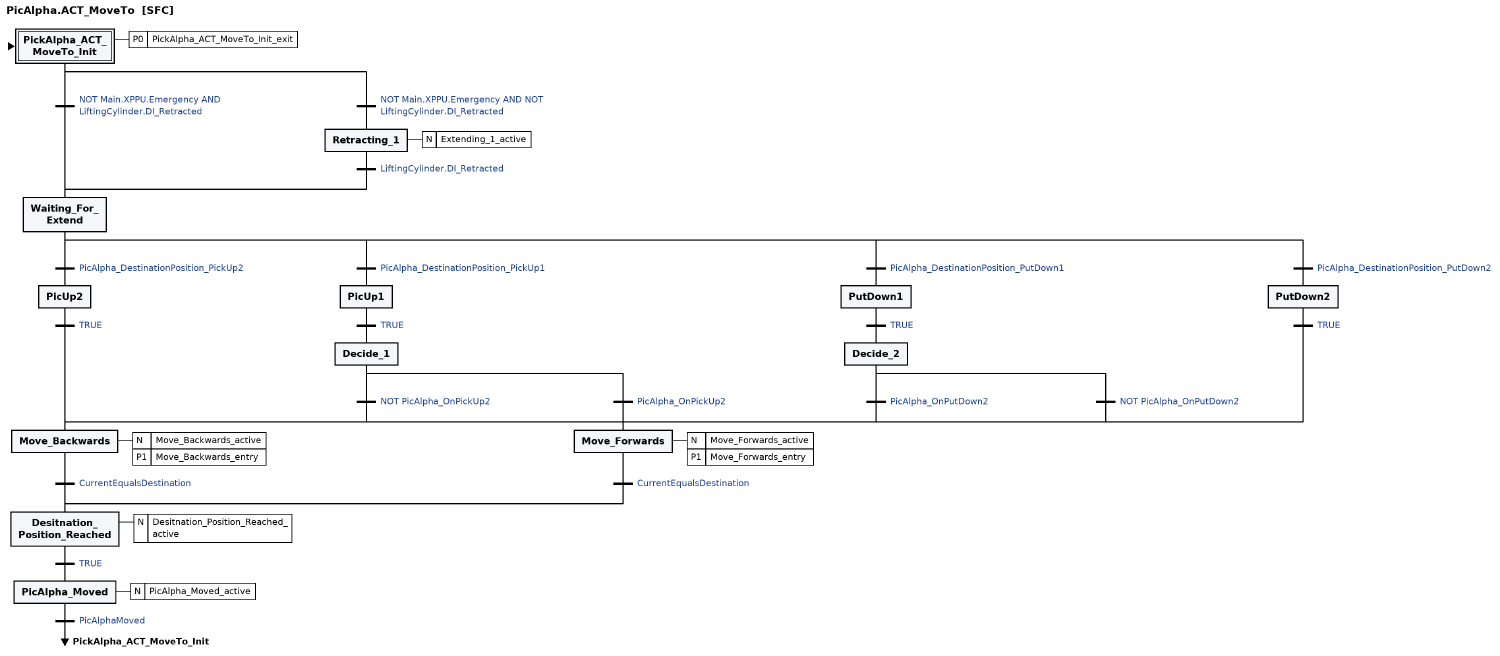
INITIAL_STEP PickAlpha_ACT_MoveTo_Init:
  PickAlpha_ACT_MoveTo_Init_exit(P0);
END_STEP
TRANSITION FROM PickAlpha_ACT_MoveTo_Init TO Waiting_For_Extend
  := NOT Main.XPPU.Emergency AND LiftingCylinder.DI_Retracted;
END_TRANSITION
TRANSITION FROM PickAlpha_ACT_MoveTo_Init TO Retracting_1
  := NOT Main.XPPU.Emergency AND NOT LiftingCylinder.DI_Retracted;
END_TRANSITION
STEP Retracting_1:
  Extending_1_active(N);
END_STEP
TRANSITION FROM Retracting_1 TO Waiting_For_Extend
  := LiftingCylinder.DI_Retracted;
END_TRANSITION
STEP Waiting_For_Extend:
END_STEP
TRANSITION FROM Waiting_For_Extend TO PicUp2
  := PicAlpha_DestinationPosition_PickUp2;
END_TRANSITION
TRANSITION FROM Waiting_For_Extend TO PicUp1
  := PicAlpha_DestinationPosition_PickUp1;
END_TRANSITION
TRANSITION FROM Waiting_For_Extend TO PutDown1
  := PicAlpha_DestinationPosition_PutDown1;
END_TRANSITION
TRANSITION FROM Waiting_For_Extend TO PutDown2
  := PicAlpha_DestinationPosition_PutDown2;
END_TRANSITION
STEP PicUp2:
END_STEP
TRANSITION FROM PicUp2 TO Move_Backwards
  := TRUE;
END_TRANSITION
STEP Move_Backwards:
  Move_Backwards_active(N);
  Move_Backwards_entry(P1);
END_STEP
TRANSITION FROM Move_Backwards TO Desitnation_Position_Reached
  := CurrentEqualsDestination;
END_TRANSITION
STEP PicUp1:
END_STEP
TRANSITION FROM PicUp1 TO Decide_1
  := TRUE;
END_TRANSITION
STEP Decide_1:
END_STEP
TRANSITION FROM Decide_1 TO Move_Backwards
  := NOT PicAlpha_OnPickUp2;
END_TRANSITION
TRANSITION FROM Decide_1 TO Move_Forwards
  := PicAlpha_OnPickUp2;
END_TRANSITION
STEP PutDown1:
END_STEP
TRANSITION FROM PutDown1 TO Decide_2
  := TRUE;
END_TRANSITION
STEP Decide_2:
END_STEP
TRANSITION FROM Decide_2 TO Move_Backwards
  := PicAlpha_OnPutDown2;
END_TRANSITION
TRANSITION FROM Decide_2 TO Move_Forwards
  := NOT PicAlpha_OnPutDown2;
END_TRANSITION
STEP PutDown2:
END_STEP
TRANSITION FROM PutDown2 TO Move_Forwards
  := TRUE;
END_TRANSITION
STEP Move_Forwards:
  Move_Forwards_active(N);
  Move_Forwards_entry(P1);
END_STEP
TRANSITION FROM Move_Forwards TO Desitnation_Position_Reached
  := CurrentEqualsDestination;
END_TRANSITION
STEP Desitnation_Position_Reached:
  Desitnation_Position_Reached_active(N);
END_STEP
TRANSITION FROM Desitnation_Position_Reached TO PicAlpha_Moved
  := TRUE;
END_TRANSITION
STEP PicAlpha_Moved:
  PicAlpha_Moved_active(N);
END_STEP
TRANSITION FROM PicAlpha_Moved TO PickAlpha_ACT_MoveTo_Init
  := PicAlphaMoved;
END_TRANSITION
END_ACTION

ACTION ACT_EmergencyStop:
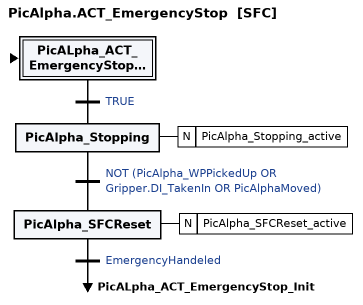
INITIAL_STEP PicALpha_ACT_EmergencyStop_Init:
END_STEP
TRANSITION FROM PicALpha_ACT_EmergencyStop_Init TO PicAlpha_Stopping
  := TRUE;
END_TRANSITION
STEP PicAlpha_Stopping:
  PicAlpha_Stopping_active(N);
END_STEP
TRANSITION FROM PicAlpha_Stopping TO PicAlpha_SFCReset
  := NOT (PicAlpha_WPPickedUp OR Gripper.DI_TakenIn OR PicAlphaMoved);
END_TRANSITION
STEP PicAlpha_SFCReset:
  PicAlpha_SFCReset_active(N);
END_STEP
TRANSITION FROM PicAlpha_SFCReset TO PicALpha_ACT_EmergencyStop_Init
  := EmergencyHandeled;
END_TRANSITION
END_ACTION

ACTION ACT_Init:
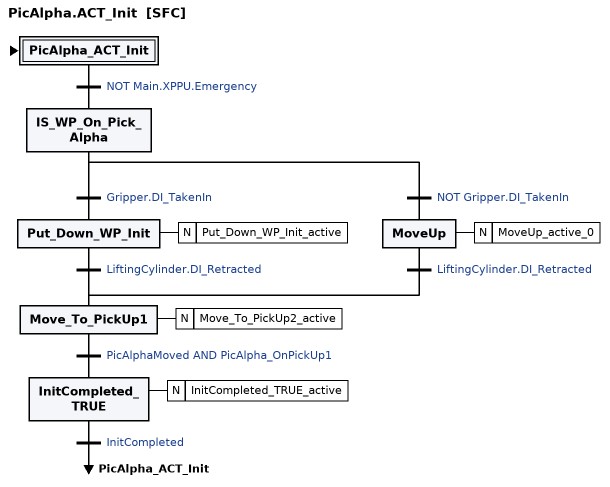
INITIAL_STEP PicAlpha_ACT_Init:
END_STEP
TRANSITION FROM PicAlpha_ACT_Init TO IS_WP_On_Pick_Alpha
  := NOT Main.XPPU.Emergency;
END_TRANSITION
STEP IS_WP_On_Pick_Alpha:
END_STEP
TRANSITION FROM IS_WP_On_Pick_Alpha TO Put_Down_WP_Init
  := Gripper.DI_TakenIn;
END_TRANSITION
TRANSITION FROM IS_WP_On_Pick_Alpha TO MoveUp
  := NOT Gripper.DI_TakenIn;
END_TRANSITION
STEP Put_Down_WP_Init:
  Put_Down_WP_Init_active(N);
END_STEP
TRANSITION FROM Put_Down_WP_Init TO Move_To_PickUp1
  := LiftingCylinder.DI_Retracted;
END_TRANSITION
STEP MoveUp:
  MoveUp_active_0(N);
END_STEP
TRANSITION FROM MoveUp TO Move_To_PickUp1
  := LiftingCylinder.DI_Retracted;
END_TRANSITION
STEP Move_To_PickUp1:
  Move_To_PickUp2_active(N);
END_STEP
TRANSITION FROM Move_To_PickUp1 TO InitCompleted_TRUE
  := PicAlphaMoved AND PicAlpha_OnPickUp1;
END_TRANSITION
STEP InitCompleted_TRUE:
  InitCompleted_TRUE_active(N);
END_STEP
TRANSITION FROM InitCompleted_TRUE TO PicAlpha_ACT_Init
  := InitCompleted;
END_TRANSITION
END_ACTION

ACTION ACT_AutomaticExecute:
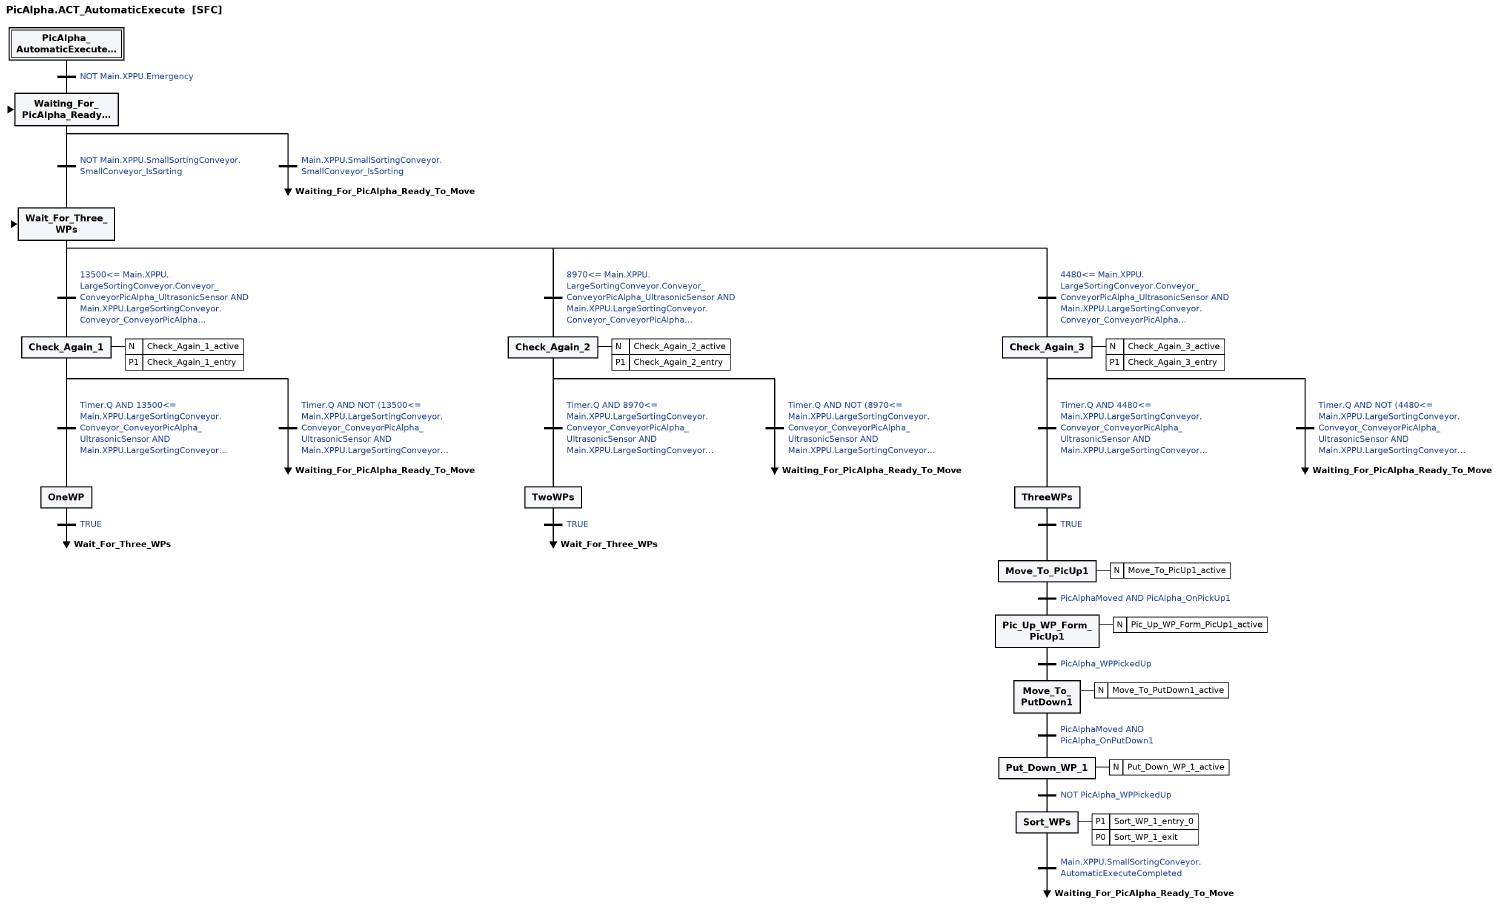
INITIAL_STEP PicAlpha_AutomaticExecute_Init:
END_STEP
TRANSITION FROM PicAlpha_AutomaticExecute_Init TO Waiting_For_PicAlpha_Ready_To_Move
  := NOT Main.XPPU.Emergency;
END_TRANSITION
STEP Waiting_For_PicAlpha_Ready_To_Move:
END_STEP
TRANSITION FROM Waiting_For_PicAlpha_Ready_To_Move TO Wait_For_Three_WPs
  := NOT Main.XPPU.SmallSortingConveyor.SmallConveyor_IsSorting;
END_TRANSITION
TRANSITION FROM Waiting_For_PicAlpha_Ready_To_Move TO Waiting_For_PicAlpha_Ready_To_Move
  := Main.XPPU.SmallSortingConveyor.SmallConveyor_IsSorting;
END_TRANSITION
STEP Wait_For_Three_WPs:
END_STEP
TRANSITION FROM Wait_For_Three_WPs TO Check_Again_1
  := 13500<= Main.XPPU.LargeSortingConveyor.Conveyor_ConveyorPicAlpha_UltrasonicSensor AND Main.XPPU.LargeSortingConveyor.Conveyor_ConveyorPicAlpha_UltrasonicSensor<=13700;
END_TRANSITION
TRANSITION FROM Wait_For_Three_WPs TO Check_Again_2
  := 8970<= Main.XPPU.LargeSortingConveyor.Conveyor_ConveyorPicAlpha_UltrasonicSensor AND Main.XPPU.LargeSortingConveyor.Conveyor_ConveyorPicAlpha_UltrasonicSensor<=9170;
END_TRANSITION
TRANSITION FROM Wait_For_Three_WPs TO Check_Again_3
  := 4480<= Main.XPPU.LargeSortingConveyor.Conveyor_ConveyorPicAlpha_UltrasonicSensor AND Main.XPPU.LargeSortingConveyor.Conveyor_ConveyorPicAlpha_UltrasonicSensor<=4680;
END_TRANSITION
STEP Check_Again_1:
  Check_Again_1_active(N);
  Check_Again_1_entry(P1);
END_STEP
TRANSITION FROM Check_Again_1 TO OneWP
  := Timer.Q AND 13500<= Main.XPPU.LargeSortingConveyor.Conveyor_ConveyorPicAlpha_UltrasonicSensor AND Main.XPPU.LargeSortingConveyor.Conveyor_ConveyorPicAlpha_UltrasonicSensor<=13700;
END_TRANSITION
TRANSITION FROM Check_Again_1 TO Waiting_For_PicAlpha_Ready_To_Move
  := Timer.Q AND NOT (13500<= Main.XPPU.LargeSortingConveyor.Conveyor_ConveyorPicAlpha_UltrasonicSensor AND Main.XPPU.LargeSortingConveyor.Conveyor_ConveyorPicAlpha_UltrasonicSensor<=13700);
END_TRANSITION
STEP OneWP:
END_STEP
TRANSITION FROM OneWP TO Wait_For_Three_WPs
  := TRUE;
END_TRANSITION
STEP Check_Again_2:
  Check_Again_2_active(N);
  Check_Again_2_entry(P1);
END_STEP
TRANSITION FROM Check_Again_2 TO TwoWPs
  := Timer.Q AND 8970<= Main.XPPU.LargeSortingConveyor.Conveyor_ConveyorPicAlpha_UltrasonicSensor AND Main.XPPU.LargeSortingConveyor.Conveyor_ConveyorPicAlpha_UltrasonicSensor<=9170;
END_TRANSITION
TRANSITION FROM Check_Again_2 TO Waiting_For_PicAlpha_Ready_To_Move
  := Timer.Q AND NOT (8970<= Main.XPPU.LargeSortingConveyor.Conveyor_ConveyorPicAlpha_UltrasonicSensor AND Main.XPPU.LargeSortingConveyor.Conveyor_ConveyorPicAlpha_UltrasonicSensor<=9170);
END_TRANSITION
STEP TwoWPs:
END_STEP
TRANSITION FROM TwoWPs TO Wait_For_Three_WPs
  := TRUE;
END_TRANSITION
STEP Check_Again_3:
  Check_Again_3_active(N);
  Check_Again_3_entry(P1);
END_STEP
TRANSITION FROM Check_Again_3 TO ThreeWPs
  := Timer.Q AND 4480<= Main.XPPU.LargeSortingConveyor.Conveyor_ConveyorPicAlpha_UltrasonicSensor AND Main.XPPU.LargeSortingConveyor.Conveyor_ConveyorPicAlpha_UltrasonicSensor<=4680;
END_TRANSITION
TRANSITION FROM Check_Again_3 TO Waiting_For_PicAlpha_Ready_To_Move
  := Timer.Q AND NOT (4480<= Main.XPPU.LargeSortingConveyor.Conveyor_ConveyorPicAlpha_UltrasonicSensor AND Main.XPPU.LargeSortingConveyor.Conveyor_ConveyorPicAlpha_UltrasonicSensor<=4680);
END_TRANSITION
STEP ThreeWPs:
END_STEP
TRANSITION FROM ThreeWPs TO Move_To_PicUp1
  := TRUE;
END_TRANSITION
STEP Move_To_PicUp1:
  Move_To_PicUp1_active(N);
END_STEP
TRANSITION FROM Move_To_PicUp1 TO Pic_Up_WP_Form_PicUp1
  := PicAlphaMoved AND PicAlpha_OnPickUp1;
END_TRANSITION
STEP Pic_Up_WP_Form_PicUp1:
  Pic_Up_WP_Form_PicUp1_active(N);
END_STEP
TRANSITION FROM Pic_Up_WP_Form_PicUp1 TO Move_To_PutDown1
  := PicAlpha_WPPickedUp;
END_TRANSITION
STEP Move_To_PutDown1:
  Move_To_PutDown1_active(N);
END_STEP
TRANSITION FROM Move_To_PutDown1 TO Put_Down_WP_1
  := PicAlphaMoved AND PicAlpha_OnPutDown1;
END_TRANSITION
STEP Put_Down_WP_1:
  Put_Down_WP_1_active(N);
END_STEP
TRANSITION FROM Put_Down_WP_1 TO Sort_WPs
  := NOT PicAlpha_WPPickedUp;
END_TRANSITION
STEP Sort_WPs:
  Sort_WP_1_entry_0(P1);
  Sort_WP_1_exit(P0);
END_STEP
TRANSITION FROM Sort_WPs TO Waiting_For_PicAlpha_Ready_To_Move
  := Main.XPPU.SmallSortingConveyor.AutomaticExecuteCompleted;
END_TRANSITION
END_ACTION

ACTION Sort_WP_1_active:
                      Main.XPPU.SmallSortingConveyor.ACT_SortWP();
                    
END_ACTION

ACTION Sort_WP_3_entry_0:
                      SC_PicAlpha_AllowToOperate:=TRUE;
                    
END_ACTION

ACTION Extending_active:
                      LiftingCylinder.ACT_Extend();
                    
END_ACTION

ACTION Check_Again_1_entry:
                      Timer(IN:=FALSE);
                    
END_ACTION

ACTION Move_Forwards_active:
                      Motor.ACT_TurnForwards();
IF(PicAlpha_DestinationPosition_PickUp2=PicAlpha_OnPickUp2 AND PicAlpha_OnPickUp2)THEN
	CurrentEqualsDestination:=TRUE;
ELSIF(PicAlpha_DestinationPosition_PutDown1=PicAlpha_OnPutDown1 AND PicAlpha_OnPutDown1 )THEN
	CurrentEqualsDestination:=TRUE;	
ELSIF(PicAlpha_DestinationPosition_PutDown2=PicAlpha_OnPutDown2 AND PicAlpha_OnPutDown2)THEN
	CurrentEqualsDestination:=TRUE;
END_IF
                    
END_ACTION

ACTION Desitnation_Position_Reached_active:
                      Motor.ACT_Stop();
                    
END_ACTION

ACTION Sort_WP_2_entry:
                      Main.XPPU.SmallSortingConveyor.HelpACT_WPSorted_FALSE();
                    
END_ACTION

ACTION Sort_WP_3_entry:
                      Main.XPPU.SmallSortingConveyor.HelpACT_WPSorted_FALSE();
                    
END_ACTION

ACTION PickAlpha_ACT_MoveTo_Init_exit:
                      PicAlphaMoved:=FALSE;
                    
END_ACTION

ACTION Sort_WP_2_active:
                      Main.XPPU.SmallSortingConveyor.ACT_SortWP();
                    
END_ACTION

ACTION Seperate_First_WP_active:
                      Main.XPPU.ConveyorPicAlpha.ACT_SeperateWP();
                    
END_ACTION

ACTION Move_To_PicUp1_active:
                      PicAlpha_DestinationPosition_PickUp1:=TRUE;
PicAlpha_DestinationPosition_PickUp2:=FALSE;
PicAlpha_DestinationPosition_PutDown1:=FALSE;
PicAlpha_DestinationPosition_PutDown2:=FALSE;
ACT_MoveTo();
                    
END_ACTION

ACTION MoveUp_active:
                      LiftingCylinder.ACT_Retract();
                    
END_ACTION

ACTION Move_Backwards_entry:
                      CurrentEqualsDestination:=FALSE;
                    
END_ACTION

ACTION Extending_1_active:
                      LiftingCylinder.ACT_Retract();
                    
END_ACTION

ACTION Retracting_PicAlpha_exit:
                      PicAlpha_WPPickedUp:=TRUE;
                    
END_ACTION

ACTION Sort_WP_2_exit:
                      SC_PicAlpha_AllowToOperate:=FALSE;
                    
END_ACTION

ACTION Sort_WP_3_exit:
                      SC_PicAlpha_AllowToOperate:=FALSE;
                    
END_ACTION

ACTION Sort_WP_2_entry_0:
                      SC_PicAlpha_AllowToOperate:=TRUE;
                    
END_ACTION

ACTION Pic_Up_WP_Form_PicUp1_active:
                      ACT_PickUpWP();
                    
END_ACTION

ACTION PicAlpha_Moved_active:
                      PicAlphaMoved:=TRUE;
                    
END_ACTION

ACTION Put_Down_WP_Init_active:
                      ACT_PutDownWP();
                    
END_ACTION

ACTION Extending_PicUp_active:
                      LiftingCylinder.ACT_Extend();
                    
END_ACTION

ACTION Check_Again_3_entry:
                      Timer(IN:=FALSE);
                    
END_ACTION

ACTION Error_active:
                      LiftingCylinder.ACT_Retract();
PicAlpha_SoftwareEmergency:=true;
                    
END_ACTION

ACTION Put_Down_WP_1_active:
                      ACT_PutDownWP();
                    
END_ACTION

ACTION Sort_WP_3_active:
                      Main.XPPU.SmallSortingConveyor.ACT_SortWP();
                    
END_ACTION

ACTION Check_Again_2_active:
                      Timer(IN:=TRUE, PT:=T#500ms);
                    
END_ACTION

ACTION Sort_WP_1_entry:
                      SC_PicAlpha_AllowToOperate:=TRUE;
                    
END_ACTION

ACTION Step0_ACT_EmergencyStop_active:
                      SFCReset:=TRUE;
                    
END_ACTION

ACTION Sort_WP_1_entry_0:
                      SC_PicAlpha_AllowToOperate:=TRUE;
                    
END_ACTION

ACTION Check_Again_3_active:
                      Timer(IN:=TRUE, PT:=T#500ms);
                    
END_ACTION

ACTION Retracting_active:
                      PicAlphaVacuumHit:=FALSE;
LiftingCylinder.ACT_Retract();
                    
END_ACTION

ACTION Move_Forwards_entry:
                      CurrentEqualsDestination:=FALSE;
                    
END_ACTION

ACTION Seperate_First_WP_entry:
                      //Main.XPPU.ConveyorPicALpha.HelpACT_WPSeperated_FALSE();
                    
END_ACTION

ACTION MoveUp_entry:
                      Timer(IN:=FALSE);
                    
END_ACTION

ACTION Retracting_exit:
                      PicAlpha_WPPickedUp:=FALSE;
                    
END_ACTION

ACTION Stop_Vacuum_active:
                      Gripper.ACT_Release();
PicAlphaVacuumHit:=TRUE;
                    
END_ACTION

ACTION Check_Again_1_active:
                      Timer(IN:=TRUE, PT:=T#500ms);
                    
END_ACTION

ACTION InitCompleted_FALSE_active:
                      InitCompleted:=FALSE;
                    
END_ACTION

ACTION Intaking_PicUp_active:
                      Gripper.ACT_Intake();
Timer(IN:=true, PT:=T#2s);
                    
END_ACTION

ACTION Retracting_PicAlpha_active:
                      LiftingCylinder.ACT_Retract();
                    
END_ACTION

ACTION PicAlpha_Stopping_active:
                      PicAlpha_WPPickedUp:=FALSE;
PicAlpha_DestinationPosition_PickUp1:=FALSE;
PicAlpha_DestinationPosition_PickUp2:=FALSE;
PicAlpha_DestinationPosition_PutDown1:=FALSE;
PicAlpha_DestinationPosition_PutDown2:=FALSE;

Gripper.ACT_Release();
PicAlphaVacuumHit:=FALSE;	
Motor.ACT_Stop();

CurrentEqualsDestination:=FALSE;
PicAlphaMoved:=FALSE;
                    
END_ACTION

ACTION PicAlpha_SFCReset_active:
                       EmergencyHandeled:=TRUE;	
                    
END_ACTION

ACTION Move_To_PutDown1_active:
                      PicAlpha_DestinationPosition_PickUp1:=FALSE;
PicAlpha_DestinationPosition_PickUp2:=FALSE;
PicAlpha_DestinationPosition_PutDown1:=TRUE;
PicAlpha_DestinationPosition_PutDown2:=FALSE;
ACT_MoveTo();
                    
END_ACTION

ACTION Seperate_Second_WP_entry:
                      //Main.XPPU.ConveyorPicALpha.HelpACT_WPSeperated_FALSE();
                    
END_ACTION

ACTION Intaking_PicUp_entry:
                      Timer(IN:=FALSE);
                    
END_ACTION

ACTION MoveUp_active_0:
                      LiftingCylinder.ACT_Retract();
                    
END_ACTION

ACTION Sort_WP_1_exit:
                      SC_PicAlpha_AllowToOperate:=FALSE;
                    
END_ACTION

ACTION InitCompleted_TRUE_active:
                      InitCompleted:=TRUE;
                    
END_ACTION

ACTION PicAlpha_StopVacuum_active:
                      Gripper.ACT_Release();
                    
END_ACTION

ACTION Seperate_Second_WP_active:
                      Main.XPPU.ConveyorPicAlpha.ACT_SeperateWP();
                    
END_ACTION

ACTION Move_Backwards_active:
                      Motor.ACT_TurnBackwards();
CurrentEqualsDestination:=FALSE;
IF(PicAlpha_DestinationPosition_PickUp1=PicAlpha_OnPickUp1 AND PicAlpha_OnPickUp1)THEN
	CurrentEqualsDestination:=TRUE;
ELSIF(PicAlpha_DestinationPosition_PickUp2=PicAlpha_OnPickUp2 AND PicAlpha_OnPickUp2)THEN
	CurrentEqualsDestination:=TRUE;
ELSIF(PicAlpha_DestinationPosition_PutDown1=PicAlpha_OnPutDown1 AND PicAlpha_OnPutDown1)THEN
	CurrentEqualsDestination:=TRUE;	
END_IF
                    
END_ACTION

ACTION Check_Again_2_entry:
                      Timer(IN:=FALSE);
                    
END_ACTION

ACTION Move_To_PickUp2_active:
                      PicAlpha_DestinationPosition_PickUp1:=TRUE;
PicAlpha_DestinationPosition_PickUp2:=FALSE;
PicAlpha_DestinationPosition_PutDown1:=FALSE;
PicAlpha_DestinationPosition_PutDown2:=FALSE;

ACT_MoveTo();
                    
END_ACTION
END_FUNCTION_BLOCK

FUNCTION_BLOCK SeperatorConveyor_Refill
VAR_INPUT	
	SwitchStopper : Switch;
	Motor : Motor;
	//Software	
	SFCReset : BOOL;
	InitCompleted : BOOL;
	LSC_AllowedToOperate : BOOL;
	AutomaticExecuteReceivingCompleted : BOOL;
	EmergencyHandeled : BOOL;
END_VAR
VAR_OUTPUT	
	//Software	
	SeperatorConveyor_WPSeperated : BOOL;
	SeperatorConveyor_IsRefilling : BOOL;
	SeperatorConveyor_RefillingIsActive : BOOL;
	SeperatorConveyor_NumberOfWPs : INT;
END_VAR
VAR
	//Hardware
	SeperaterConveyor_Beginning_PresenceSensor AT %I* : BOOL;
	SeperaterConveyor_End_PresenceSensor AT %I* : BOOL;
	
	//Software
	Timer:TON;
END_VAR

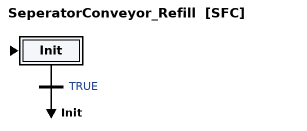
INITIAL_STEP Init:
END_STEP
TRANSITION FROM Init TO Init
  := TRUE;
END_TRANSITION

ACTION Turn_On_Conveyor_entry:
                      Timer(IN:=FALSE);
                    
END_ACTION

ACTION HelpACT_WPSeperated_FALSE:
                      SeperatorConveyor_WPSeperated:=FALSE;
                    
END_ACTION

ACTION TurnForwards_PAC_entry:
                      Timer(IN:=FALSE);
                    
END_ACTION

ACTION Turn_Off_Conveyor_active_0:
                      Motor.ACT_Stop();
                    
END_ACTION

ACTION Stop_PAC_active:
                      Motor.ACT_Stop();
                    
END_ACTION

ACTION Turn_On_Conveyor_active:
                      Motor.ACT_TurnForwards();

Timer(IN:=TRUE, PT:=T#500ms);
	
                    
END_ACTION

ACTION Refilling_LargeSortingConveyor_entry:
                      SeperatorConveyor_IsRefilling:=TRUE;
SeperatorConveyor_RefillingIsActive:=TRUE;
                    
END_ACTION

ACTION SeperaterConveyor_SFCReset_active:
                      EmergencyHandeled:=TRUE;		
                    
END_ACTION

ACTION Stop_Conveyor_active:
                      Motor.ACT_Stop();	
                    
END_ACTION

ACTION Trun_Forwards_AE_entry:
                      Timer(IN:=FALSE);
                    
END_ACTION

ACTION Sort_WP_active_0:
                      Main.XPPU.LargeSortingConveyor.ACT_SortWP();
                    
END_ACTION

ACTION Count_Up_active_0:
                      SeperatorConveyor_NumberOfWPs:=SeperatorConveyor_NumberOfWPs+1;
                    
END_ACTION

ACTION All_WPs_Refilled_active:
                      SeperatorConveyor_RefillingIsActive:=FALSE;
                    
END_ACTION

ACTION Short_Delay_entry_0:
                      Timer(IN:=FALSE);
AutomaticExecuteReceivingCompleted:=FALSE;
                    
END_ACTION

ACTION Turn_Off_Conveyor_entry:
                      Timer(IN:=FALSE);
                    
END_ACTION

ACTION Turn_On_Conveyor_exit:
                      SeperatorConveyor_NumberOfWPs:=SeperatorConveyor_NumberOfWPs - 1;
                    
END_ACTION

ACTION Seperate_WP_entry:
                      SeperatorConveyor_WPSeperated:=FALSE;
                    
END_ACTION

ACTION Count_Up_active:
                      SeperatorConveyor_NumberOfWPs:=SeperatorConveyor_NumberOfWPs+1;
                    
END_ACTION

ACTION Stop_Conveyor_Init_active:
                      Motor.ACT_Stop();
                    
END_ACTION

ACTION WP_Refilled_active:
                      SeperatorConveyor_IsRefilling:=FALSE;
                    
END_ACTION

ACTION Turn_Forwards_entry:
                      Timer(IN:=FALSE);
                    
END_ACTION

ACTION SeperatorConveyor_ACT_AutomaticExecute_Init_entry:
                      
                    
END_ACTION

ACTION Stop_Conveyor_Init_exit:
                      InitCompleted:=TRUE;
                    
END_ACTION

ACTION Turn_Off_Conveyor_2_active:
                      Motor.ACT_Stop();
SeperatorConveyor_WPSeperated:=TRUE;
                    
END_ACTION

ACTION Short_Delay_For_Only_One_Count_entry:
                      Timer(IN:=FALSE);
                    
END_ACTION

ACTION Sort_WP_active:
                      Main.XPPU.LargeSortingConveyor.ACT_SortWP();
                    
END_ACTION

ACTION Trun_Forwards_AE_active:
                      Motor.ACT_TurnForwards();
Timer(IN:=TRUE, PT:=T#2000ms);
                    
END_ACTION

ACTION Refillinf_LargeSortingConveyor_entry:
                      SeperatorConveyor_IsRefilling:=TRUE;
                    
END_ACTION

ACTION Switch_Retracting_active:
                      SwitchStopper.ACT_Retract();
                    
END_ACTION

ACTION Turn_Forwards_active:
                      Motor.ACT_TurnForwards();
Timer(IN:=TRUE, PT:=T#1500ms);
                    
END_ACTION

ACTION Short_Delay_PACReceiving_active:
                      Timer(IN:=TRUE, PT:=T#500ms);
                    
END_ACTION

ACTION Move_PCA_Forward_active:
                      Motor.ACT_TurnForwards();
Timer(IN:=TRUE, PT:=T#3000ms);
                    
END_ACTION

ACTION Count_Up_active_1:
                      SeperatorConveyor_NumberOfWPs:=SeperatorConveyor_NumberOfWPs+1;
                    
END_ACTION

ACTION Extend_Switch_active_0:
                      SwitchStopper.ACT_Retract();
                    
END_ACTION

ACTION Sort_WP_entry_0:
                      LSC_AllowedToOperate:=TRUE;
                    
END_ACTION

ACTION Turn_Conveyor_On_active:
                      SeperatorConveyor_WPSeperated:=FALSE;
Motor.ACT_TurnForwards();
                    
END_ACTION

ACTION Refilling_Sorting_Conveyor_entry:
                      SeperatorConveyor_IsRefilling:=TRUE;
                    
END_ACTION

ACTION Short_Delay_active:
                      Timer(IN:=TRUE, PT:=T#500ms);
                    
END_ACTION

ACTION Retract_Switch_active:
                      SwitchStopper.ACT_Retract();
                    
END_ACTION

ACTION ResetRunning_PACReceiving_active:
                      AutomaticExecuteReceivingCompleted:=TRUE;
                    
END_ACTION

ACTION Seperate_WP_active:
                      SeperatorConveyor_IsRefilling:=TRUE;
SeperatorConveyor_WPSeperated:=FALSE;
ACT_SeperateWP();
                    
END_ACTION

ACTION Short_Delay_PACReceiving_entry:
                      Timer(IN:=FALSE);
                    
END_ACTION

ACTION Short_Delay_For_Only_One_Count_active:
                      Timer(IN:=TRUE, PT:=T#500ms);
                    
END_ACTION

ACTION Sort_WP_exit:
                      
                    
END_ACTION

ACTION Refilling_Sorting_Conveyor_active:
                      ACT_Refill();
                    
END_ACTION

ACTION Extend_Switch_exit:
                      
                    
END_ACTION

ACTION Short_Delay_entry:
                      Timer(IN:=FALSE);
                    
END_ACTION

ACTION Sort_WP_entry:
                      Main.XPPU.LargeSortingConveyor.HelpACT_ConveyorWPSortet_FALSE();
                    
END_ACTION

ACTION Conveyor_Stopping_active:
                      SeperatorConveyor_WPSeperated:=FALSE;
SeperatorConveyor_IsRefilling:=FALSE;
SeperatorConveyor_NumberOfWPs:=0;

Motor.ACT_Stop();
                    
END_ACTION

ACTION Sort_WP_exit_0:
                      LSC_AllowedToOperate:=FALSE;
                    
END_ACTION

ACTION Turn_Off_Conveyor_active:
                      Timer(IN:=TRUE, PT:=T#500ms);
                    
END_ACTION

ACTION Refillinf_LargeSortingConveyor_active:
                      ACT_Refill();
                    
END_ACTION

ACTION Refilling_LargeSortingConveyor_active:
                      ACT_Refill();
                    
END_ACTION

ACTION Extend_Switch_active:
                      SwitchStopper.ACT_Extend();
                    
END_ACTION

ACTION Short_Delay_active_0:
                      Timer(IN:=TRUE, PT:=T#200ms);
                    
END_ACTION

ACTION Extend_Switch_To_Seperate_active:
                      SwitchStopper.ACT_Extend();
                    
END_ACTION

ACTION ACT_AutomaticExecute:
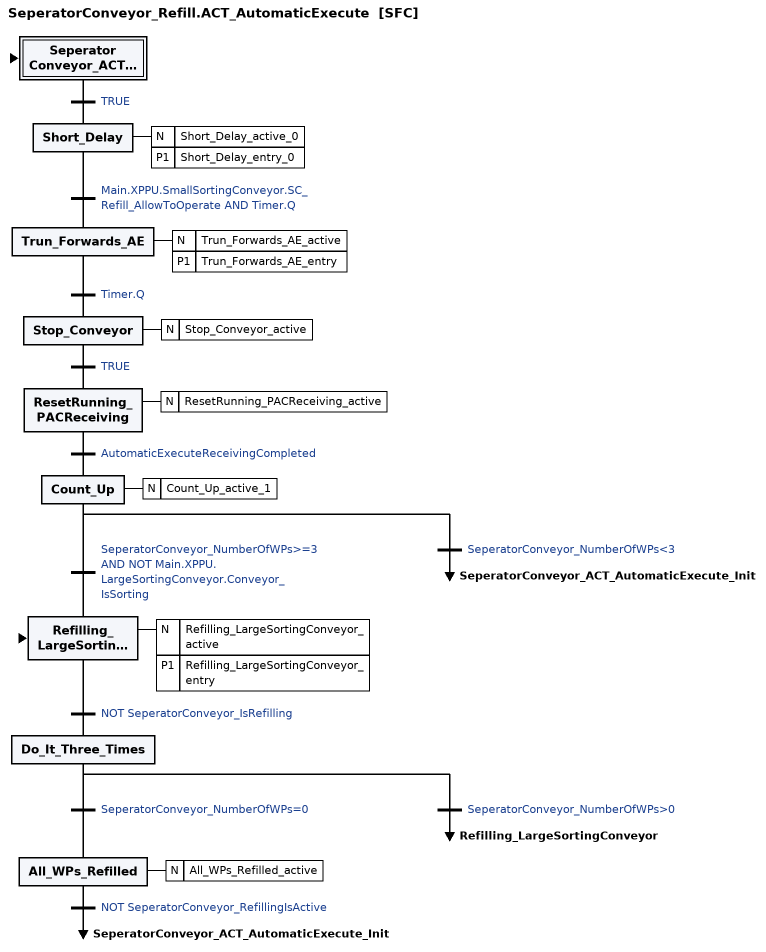
INITIAL_STEP SeperatorConveyor_ACT_AutomaticExecute_Init:
END_STEP
TRANSITION FROM SeperatorConveyor_ACT_AutomaticExecute_Init TO Short_Delay
  := TRUE;
END_TRANSITION
STEP Short_Delay:
  Short_Delay_active_0(N);
  Short_Delay_entry_0(P1);
END_STEP
TRANSITION FROM Short_Delay TO Trun_Forwards_AE
  := Main.XPPU.SmallSortingConveyor.SC_Refill_AllowToOperate AND Timer.Q;
END_TRANSITION
STEP Trun_Forwards_AE:
  Trun_Forwards_AE_active(N);
  Trun_Forwards_AE_entry(P1);
END_STEP
TRANSITION FROM Trun_Forwards_AE TO Stop_Conveyor
  := Timer.Q;
END_TRANSITION
STEP Stop_Conveyor:
  Stop_Conveyor_active(N);
END_STEP
TRANSITION FROM Stop_Conveyor TO ResetRunning_PACReceiving
  := TRUE;
END_TRANSITION
STEP ResetRunning_PACReceiving:
  ResetRunning_PACReceiving_active(N);
END_STEP
TRANSITION FROM ResetRunning_PACReceiving TO Count_Up
  := AutomaticExecuteReceivingCompleted;
END_TRANSITION
STEP Count_Up:
  Count_Up_active_1(N);
END_STEP
TRANSITION FROM Count_Up TO Refilling_LargeSortingConveyor
  := SeperatorConveyor_NumberOfWPs>=3 AND NOT Main.XPPU.LargeSortingConveyor.Conveyor_IsSorting;
END_TRANSITION
TRANSITION FROM Count_Up TO SeperatorConveyor_ACT_AutomaticExecute_Init
  := SeperatorConveyor_NumberOfWPs<3;
END_TRANSITION
STEP Refilling_LargeSortingConveyor:
  Refilling_LargeSortingConveyor_active(N);
  Refilling_LargeSortingConveyor_entry(P1);
END_STEP
TRANSITION FROM Refilling_LargeSortingConveyor TO Do_It_Three_Times
  := NOT SeperatorConveyor_IsRefilling;
END_TRANSITION
STEP Do_It_Three_Times:
END_STEP
TRANSITION FROM Do_It_Three_Times TO All_WPs_Refilled
  := SeperatorConveyor_NumberOfWPs=0;
END_TRANSITION
TRANSITION FROM Do_It_Three_Times TO Refilling_LargeSortingConveyor
  := SeperatorConveyor_NumberOfWPs>0;
END_TRANSITION
STEP All_WPs_Refilled:
  All_WPs_Refilled_active(N);
END_STEP
TRANSITION FROM All_WPs_Refilled TO SeperatorConveyor_ACT_AutomaticExecute_Init
  := NOT SeperatorConveyor_RefillingIsActive;
END_TRANSITION
END_ACTION

ACTION ACT_EmergencyStop:
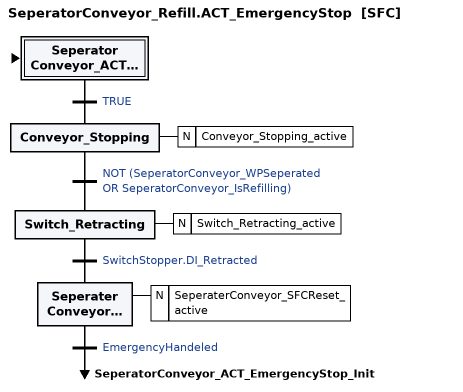
INITIAL_STEP SeperatorConveyor_ACT_EmergencyStop_Init:
END_STEP
TRANSITION FROM SeperatorConveyor_ACT_EmergencyStop_Init TO Conveyor_Stopping
  := TRUE;
END_TRANSITION
STEP Conveyor_Stopping:
  Conveyor_Stopping_active(N);
END_STEP
TRANSITION FROM Conveyor_Stopping TO Switch_Retracting
  := NOT (SeperatorConveyor_WPSeperated OR SeperatorConveyor_IsRefilling);
END_TRANSITION
STEP Switch_Retracting:
  Switch_Retracting_active(N);
END_STEP
TRANSITION FROM Switch_Retracting TO SeperaterConveyor_SFCReset
  := SwitchStopper.DI_Retracted;
END_TRANSITION
STEP SeperaterConveyor_SFCReset:
  SeperaterConveyor_SFCReset_active(N);
END_STEP
TRANSITION FROM SeperaterConveyor_SFCReset TO SeperatorConveyor_ACT_EmergencyStop_Init
  := EmergencyHandeled;
END_TRANSITION
END_ACTION

ACTION ACT_Init:
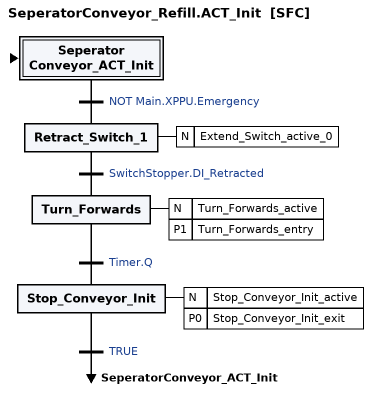
INITIAL_STEP SeperatorConveyor_ACT_Init:
END_STEP
TRANSITION FROM SeperatorConveyor_ACT_Init TO Retract_Switch_1
  := NOT Main.XPPU.Emergency;
END_TRANSITION
STEP Retract_Switch_1:
  Extend_Switch_active_0(N);
END_STEP
TRANSITION FROM Retract_Switch_1 TO Turn_Forwards
  := SwitchStopper.DI_Retracted;
END_TRANSITION
STEP Turn_Forwards:
  Turn_Forwards_active(N);
  Turn_Forwards_entry(P1);
END_STEP
TRANSITION FROM Turn_Forwards TO Stop_Conveyor_Init
  := Timer.Q;
END_TRANSITION
STEP Stop_Conveyor_Init:
  Stop_Conveyor_Init_active(N);
  Stop_Conveyor_Init_exit(P0);
END_STEP
TRANSITION FROM Stop_Conveyor_Init TO SeperatorConveyor_ACT_Init
  := TRUE;
END_TRANSITION
END_ACTION

ACTION ACT_SeperateWP:
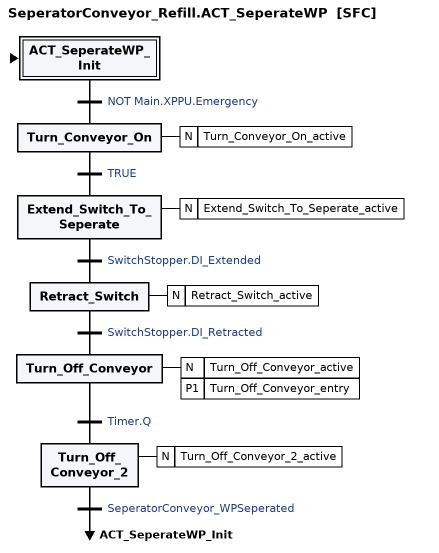
INITIAL_STEP ACT_SeperateWP_Init:
END_STEP
TRANSITION FROM ACT_SeperateWP_Init TO Turn_Conveyor_On
  := NOT Main.XPPU.Emergency;
END_TRANSITION
STEP Turn_Conveyor_On:
  Turn_Conveyor_On_active(N);
END_STEP
TRANSITION FROM Turn_Conveyor_On TO Extend_Switch_To_Seperate
  := TRUE;
END_TRANSITION
STEP Extend_Switch_To_Seperate:
  Extend_Switch_To_Seperate_active(N);
END_STEP
TRANSITION FROM Extend_Switch_To_Seperate TO Retract_Switch
  := SwitchStopper.DI_Extended;
END_TRANSITION
STEP Retract_Switch:
  Retract_Switch_active(N);
END_STEP
TRANSITION FROM Retract_Switch TO Turn_Off_Conveyor
  := SwitchStopper.DI_Retracted;
END_TRANSITION
STEP Turn_Off_Conveyor:
  Turn_Off_Conveyor_active(N);
  Turn_Off_Conveyor_entry(P1);
END_STEP
TRANSITION FROM Turn_Off_Conveyor TO Turn_Off_Conveyor_2
  := Timer.Q;
END_TRANSITION
STEP Turn_Off_Conveyor_2:
  Turn_Off_Conveyor_2_active(N);
END_STEP
TRANSITION FROM Turn_Off_Conveyor_2 TO ACT_SeperateWP_Init
  := SeperatorConveyor_WPSeperated;
END_TRANSITION
END_ACTION

ACTION ACT_Refill:
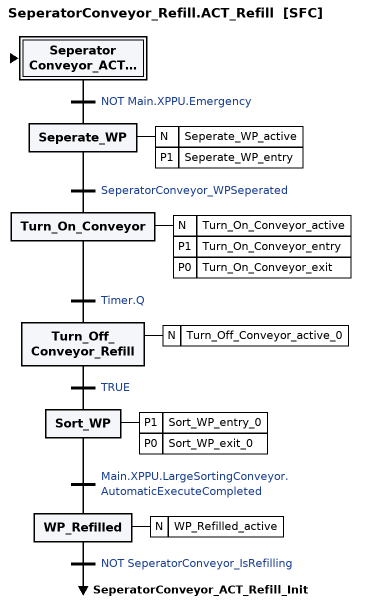
INITIAL_STEP SeperatorConveyor_ACT_Refill_Init:
END_STEP
TRANSITION FROM SeperatorConveyor_ACT_Refill_Init TO Seperate_WP
  := NOT Main.XPPU.Emergency;
END_TRANSITION
STEP Seperate_WP:
  Seperate_WP_active(N);
  Seperate_WP_entry(P1);
END_STEP
TRANSITION FROM Seperate_WP TO Turn_On_Conveyor
  := SeperatorConveyor_WPSeperated;
END_TRANSITION
STEP Turn_On_Conveyor:
  Turn_On_Conveyor_active(N);
  Turn_On_Conveyor_entry(P1);
  Turn_On_Conveyor_exit(P0);
END_STEP
TRANSITION FROM Turn_On_Conveyor TO Turn_Off_Conveyor_Refill
  := Timer.Q;
END_TRANSITION
STEP Turn_Off_Conveyor_Refill:
  Turn_Off_Conveyor_active_0(N);
END_STEP
TRANSITION FROM Turn_Off_Conveyor_Refill TO Sort_WP
  := TRUE;
END_TRANSITION
STEP Sort_WP:
  Sort_WP_entry_0(P1);
  Sort_WP_exit_0(P0);
END_STEP
TRANSITION FROM Sort_WP TO WP_Refilled
  := Main.XPPU.LargeSortingConveyor.AutomaticExecuteCompleted;
END_TRANSITION
STEP WP_Refilled:
  WP_Refilled_active(N);
END_STEP
TRANSITION FROM WP_Refilled TO SeperatorConveyor_ACT_Refill_Init
  := NOT SeperatorConveyor_IsRefilling;
END_TRANSITION
END_ACTION
END_FUNCTION_BLOCK

FUNCTION_BLOCK SeperatorConveyor_PicAlpha
VAR_INPUT	
	SwitchStopper : Switch;
	Motor : Motor;
	//Software	
	SFCReset : BOOL;
	InitCompleted : BOOL;
	SSC_AllowToOperate : BOOL; //SSC=SmallSortingConveyor
	AutomaticExecuteSendingCompleted : BOOL;
	AutomaticExecuteReceivingCompleted : BOOL;	
	EmergencyHandeled : BOOL;
END_VAR
VAR_OUTPUT	
	//Software	
	SeperaterConveyor_WPSeperated : BOOL;
END_VAR
VAR
	//Hardware
	SeperaterConveyor_Beginning_PresenceSensor AT %I* : BOOL;
	SeperaterConveyor_End_PresenceSensor AT %I* : BOOL;
	
	//Software
	Timer:TON;
END_VAR

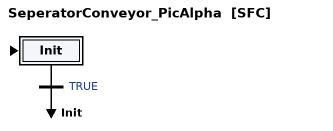
INITIAL_STEP Init:
END_STEP
TRANSITION FROM Init TO Init
  := TRUE;
END_TRANSITION

ACTION ACT_AutomaticExecute:
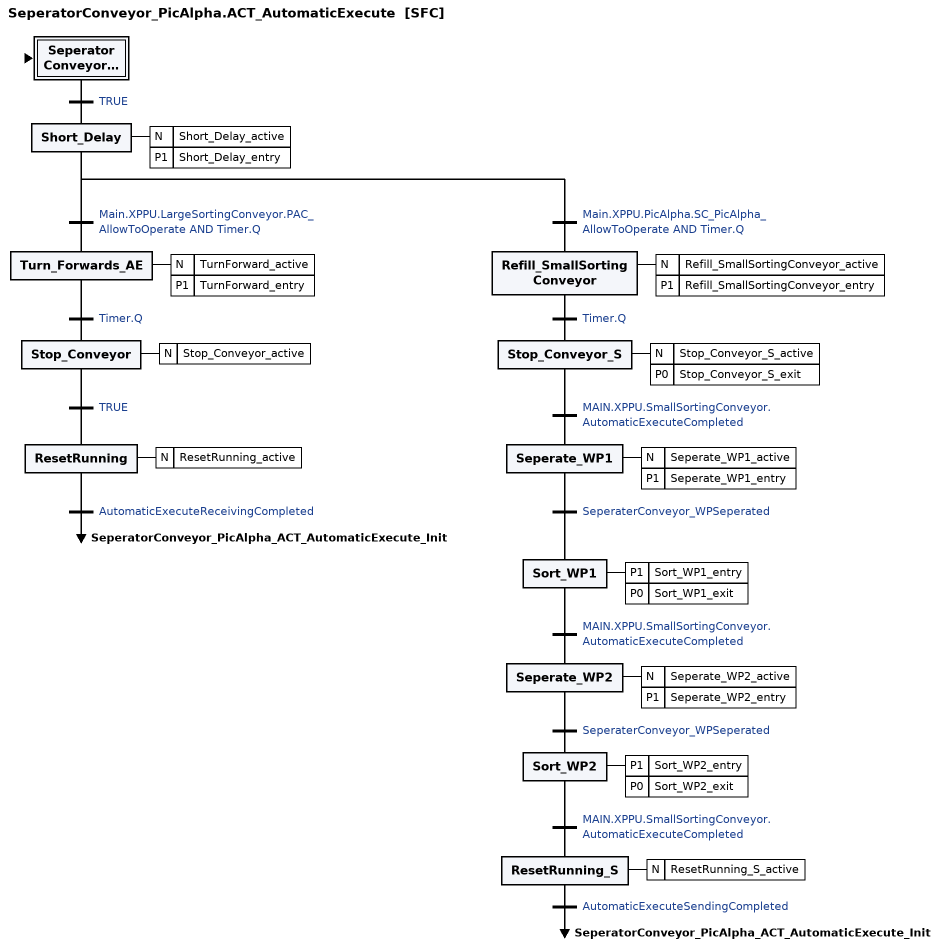
INITIAL_STEP SeperatorConveyor_PicAlpha_ACT_AutomaticExecute_Init:
END_STEP
TRANSITION FROM SeperatorConveyor_PicAlpha_ACT_AutomaticExecute_Init TO Short_Delay
  := TRUE;
END_TRANSITION
STEP Short_Delay:
  Short_Delay_active(N);
  Short_Delay_entry(P1);
END_STEP
TRANSITION FROM Short_Delay TO Turn_Forwards_AE
  := Main.XPPU.LargeSortingConveyor.PAC_AllowToOperate AND Timer.Q;
END_TRANSITION
TRANSITION FROM Short_Delay TO Refill_SmallSortingConveyor
  := Main.XPPU.PicAlpha.SC_PicAlpha_AllowToOperate AND Timer.Q;
END_TRANSITION
STEP Turn_Forwards_AE:
  TurnForward_active(N);
  TurnForward_entry(P1);
END_STEP
TRANSITION FROM Turn_Forwards_AE TO Stop_Conveyor
  := Timer.Q;
END_TRANSITION
STEP Stop_Conveyor:
  Stop_Conveyor_active(N);
END_STEP
TRANSITION FROM Stop_Conveyor TO ResetRunning
  := TRUE;
END_TRANSITION
STEP ResetRunning:
  ResetRunning_active(N);
END_STEP
TRANSITION FROM ResetRunning TO SeperatorConveyor_PicAlpha_ACT_AutomaticExecute_Init
  := AutomaticExecuteReceivingCompleted;
END_TRANSITION
STEP Refill_SmallSortingConveyor:
  Refill_SmallSortingConveyor_active(N);
  Refill_SmallSortingConveyor_entry(P1);
END_STEP
TRANSITION FROM Refill_SmallSortingConveyor TO Stop_Conveyor_S
  := Timer.Q;
END_TRANSITION
STEP Stop_Conveyor_S:
  Stop_Conveyor_S_active(N);
  Stop_Conveyor_S_exit(P0);
END_STEP
TRANSITION FROM Stop_Conveyor_S TO Seperate_WP1
  := MAIN.XPPU.SmallSortingConveyor.AutomaticExecuteCompleted;
END_TRANSITION
STEP Seperate_WP1:
  Seperate_WP1_active(N);
  Seperate_WP1_entry(P1);
END_STEP
TRANSITION FROM Seperate_WP1 TO Sort_WP1
  := SeperaterConveyor_WPSeperated;
END_TRANSITION
STEP Sort_WP1:
  Sort_WP1_entry(P1);
  Sort_WP1_exit(P0);
END_STEP
TRANSITION FROM Sort_WP1 TO Seperate_WP2
  := MAIN.XPPU.SmallSortingConveyor.AutomaticExecuteCompleted;
END_TRANSITION
STEP Seperate_WP2:
  Seperate_WP2_active(N);
  Seperate_WP2_entry(P1);
END_STEP
TRANSITION FROM Seperate_WP2 TO Sort_WP2
  := SeperaterConveyor_WPSeperated;
END_TRANSITION
STEP Sort_WP2:
  Sort_WP2_entry(P1);
  Sort_WP2_exit(P0);
END_STEP
TRANSITION FROM Sort_WP2 TO ResetRunning_S
  := MAIN.XPPU.SmallSortingConveyor.AutomaticExecuteCompleted;
END_TRANSITION
STEP ResetRunning_S:
  ResetRunning_S_active(N);
END_STEP
TRANSITION FROM ResetRunning_S TO SeperatorConveyor_PicAlpha_ACT_AutomaticExecute_Init
  := AutomaticExecuteSendingCompleted;
END_TRANSITION
END_ACTION

ACTION ACT_Init:
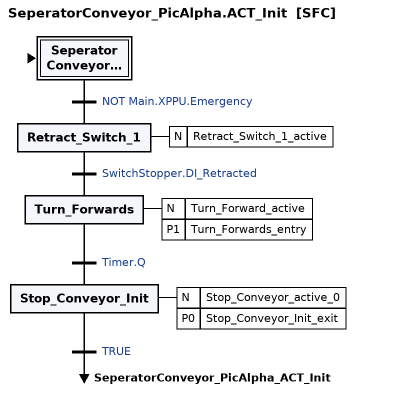
INITIAL_STEP SeperatorConveyor_PicAlpha_ACT_Init:
END_STEP
TRANSITION FROM SeperatorConveyor_PicAlpha_ACT_Init TO Retract_Switch_1
  := NOT Main.XPPU.Emergency;
END_TRANSITION
STEP Retract_Switch_1:
  Retract_Switch_1_active(N);
END_STEP
TRANSITION FROM Retract_Switch_1 TO Turn_Forwards
  := SwitchStopper.DI_Retracted;
END_TRANSITION
STEP Turn_Forwards:
  Turn_Forward_active(N);
  Turn_Forwards_entry(P1);
END_STEP
TRANSITION FROM Turn_Forwards TO Stop_Conveyor_Init
  := Timer.Q;
END_TRANSITION
STEP Stop_Conveyor_Init:
  Stop_Conveyor_active_0(N);
  Stop_Conveyor_Init_exit(P0);
END_STEP
TRANSITION FROM Stop_Conveyor_Init TO SeperatorConveyor_PicAlpha_ACT_Init
  := TRUE;
END_TRANSITION
END_ACTION

ACTION ACT_EmergencyStop:
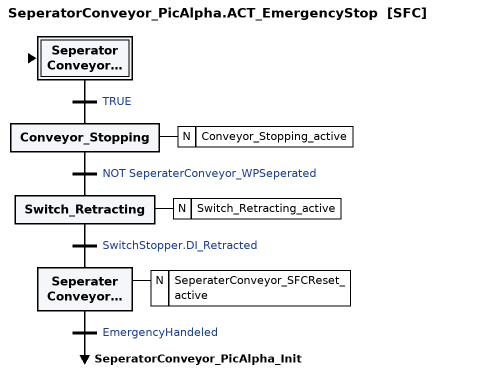
INITIAL_STEP SeperatorConveyor_PicAlpha_Init:
END_STEP
TRANSITION FROM SeperatorConveyor_PicAlpha_Init TO Conveyor_Stopping
  := TRUE;
END_TRANSITION
STEP Conveyor_Stopping:
  Conveyor_Stopping_active(N);
END_STEP
TRANSITION FROM Conveyor_Stopping TO Switch_Retracting
  := NOT SeperaterConveyor_WPSeperated;
END_TRANSITION
STEP Switch_Retracting:
  Switch_Retracting_active(N);
END_STEP
TRANSITION FROM Switch_Retracting TO SeperaterConveyor_SFCReset
  := SwitchStopper.DI_Retracted;
END_TRANSITION
STEP SeperaterConveyor_SFCReset:
  SeperaterConveyor_SFCReset_active(N);
END_STEP
TRANSITION FROM SeperaterConveyor_SFCReset TO SeperatorConveyor_PicAlpha_Init
  := EmergencyHandeled;
END_TRANSITION
END_ACTION

ACTION ACT_SeperateWP:
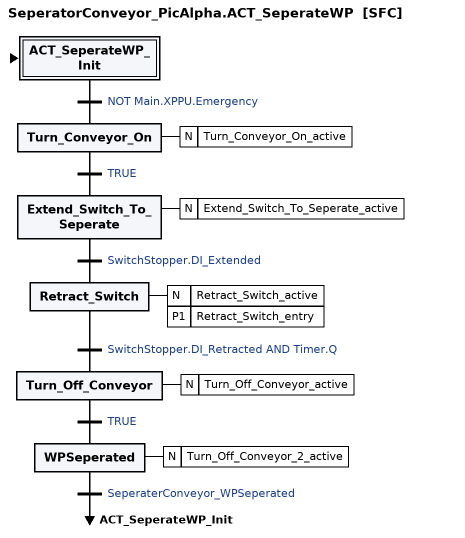
INITIAL_STEP ACT_SeperateWP_Init:
END_STEP
TRANSITION FROM ACT_SeperateWP_Init TO Turn_Conveyor_On
  := NOT Main.XPPU.Emergency;
END_TRANSITION
STEP Turn_Conveyor_On:
  Turn_Conveyor_On_active(N);
END_STEP
TRANSITION FROM Turn_Conveyor_On TO Extend_Switch_To_Seperate
  := TRUE;
END_TRANSITION
STEP Extend_Switch_To_Seperate:
  Extend_Switch_To_Seperate_active(N);
END_STEP
TRANSITION FROM Extend_Switch_To_Seperate TO Retract_Switch
  := SwitchStopper.DI_Extended;
END_TRANSITION
STEP Retract_Switch:
  Retract_Switch_active(N);
  Retract_Switch_entry(P1);
END_STEP
TRANSITION FROM Retract_Switch TO Turn_Off_Conveyor
  := SwitchStopper.DI_Retracted AND Timer.Q;
END_TRANSITION
STEP Turn_Off_Conveyor:
  Turn_Off_Conveyor_active(N);
END_STEP
TRANSITION FROM Turn_Off_Conveyor TO WPSeperated
  := TRUE;
END_TRANSITION
STEP WPSeperated:
  Turn_Off_Conveyor_2_active(N);
END_STEP
TRANSITION FROM WPSeperated TO ACT_SeperateWP_Init
  := SeperaterConveyor_WPSeperated;
END_TRANSITION
END_ACTION

ACTION Turn_Off_Conveyor_2_active:
                      SeperaterConveyor_WPSeperated:=TRUE;
                    
END_ACTION

ACTION Seperate_WP2_active:
                      ACT_SeperateWP();
                    
END_ACTION

ACTION Turn_Off_Conveyor_active:
                      Motor.ACT_Stop();
                    
END_ACTION

ACTION Turn_Conveyor_On_active:
                      SeperaterConveyor_WPSeperated:=FALSE;

Motor.ACT_TurnForwards();
                    
END_ACTION

ACTION Sort_WP1_exit:
                      SSC_AllowToOperate:=FALSE;
                    
END_ACTION

ACTION Switch_Retracting_active:
                      SwitchStopper.ACT_Retract();
                    
END_ACTION

ACTION ResetRunning_active:
                      AutomaticExecuteReceivingCompleted:=TRUE;
                    
END_ACTION

ACTION TurnForward_entry:
                      AutomaticExecuteReceivingCompleted:=FALSE;
Timer(IN:=FALSE);
                    
END_ACTION

ACTION Short_Delay_entry:
                      Timer(IN:=FALSE);
AutomaticExecuteReceivingCompleted:=FALSE;
AutomaticExecuteSendingCompleted:=FALSE;
                    
END_ACTION

ACTION Short_Delay_active:
                      Timer(IN:=TRUE, PT:=T#200ms);
                    
END_ACTION

ACTION WP_Seperated_active:
                      //SeperaterConveyor_IsRefilling:=TRUE;
                    
END_ACTION

ACTION Seperate_WP_entry:
                      SeperaterConveyor_WPSeperated:=FALSE;
                    
END_ACTION

ACTION Seperate_WP2_entry:
                      SeperaterConveyor_WPSeperated:=FALSE;
                    
END_ACTION

ACTION Refill_SmallSortingConveyor_entry:
                      AutomaticExecuteSendingCompleted:=FALSE;
Timer(IN:=FALSE);
                    
END_ACTION

ACTION Refill_SmallSortingConveyor_active:
                      Timer(IN:=TRUE, PT:=T#1000ms);
Motor.ACT_TurnForwards();
                    
END_ACTION

ACTION Retract_Switch_1_active:
                      SwitchStopper.ACT_Retract();
                    
END_ACTION

ACTION Seperate_WP_active:
                      ACT_SeperateWP();
                    
END_ACTION

ACTION Turn_Forward_active:
                      Motor.ACT_TurnForwards();
Timer(IN:=TRUE, PT:=T#2000ms);
                    
END_ACTION

ACTION Retract_Switch_entry:
                      Timer(IN:=FALSE);
                    
END_ACTION

ACTION Stop_Conveyor_S_active:
                      Motor.ACT_Stop();
SSC_AllowToOperate:=TRUE;
                    
END_ACTION

ACTION ResetRunning_S_active:
                      AutomaticExecuteSendingCompleted:=TRUE;
                    
END_ACTION

ACTION SeperaterConveyor_SFCReset_active:
                      EmergencyHandeled:=TRUE;		
                    
END_ACTION

ACTION Stop_Conveyor_Init_exit:
                      InitCompleted:=TRUE;
                    
END_ACTION

ACTION Extend_Switch_To_Seperate_active:
                      SwitchStopper.ACT_Extend();
                    
END_ACTION

ACTION Turn_On_Conveyor_entry:
                      Timer(IN:=FALSE);
                    
END_ACTION

ACTION Sort_WP1_entry:
                      SSC_AllowToOperate:=TRUE;
                    
END_ACTION

ACTION TurnForward_active:
                      Motor.ACT_TurnForwards();
Timer(IN:=TRUE, PT:=T#2000ms);
                    
END_ACTION

ACTION Stop_Conveyor_S_exit:
                      SSC_AllowToOperate:=FALSE;
                    
END_ACTION

ACTION Turn_Off_Conveyor_entry:
                      Timer(IN:=FALSE);
                    
END_ACTION

ACTION Sort_WP2_entry:
                      SSC_AllowToOperate:=TRUE;
                    
END_ACTION

ACTION Conveyor_Stopping_active:
                      SeperaterConveyor_WPSeperated:=FALSE;
Motor.ACT_Stop();
                    
END_ACTION

ACTION Retract_Switch_active:
                      SwitchStopper.ACT_Retract();
Timer(IN:=TRUE, PT:=T#1500ms);
                    
END_ACTION

ACTION Seperate_WP1_active:
                      ACT_SeperateWP();
                    
END_ACTION

ACTION Turn_Forwards_entry:
                      Timer(IN:=FALSE);
                    
END_ACTION

ACTION Stop_Conveyor_active:
                      Motor.ACT_Stop();
                    
END_ACTION

ACTION Turn_Off_Conveyor_active_0:
                      Motor.ACT_Stop();
                    
END_ACTION

ACTION Sort_WP2_exit:
                      SSC_AllowToOperate:=FALSE;
                    
END_ACTION

ACTION Turn_On_Conveyor_active:
                      Motor.ACT_TurnForwards();

Timer(IN:=TRUE, PT:=T#2000ms);
	
                    
END_ACTION

ACTION Seperate_WP1_entry:
                      SeperaterConveyor_WPSeperated:=FALSE;
                    
END_ACTION

ACTION Retract_Switch_1_exit:
                      
                    
END_ACTION

ACTION Stop_Conveyor_active_0:
                      Motor.ACT_Stop();
                    
END_ACTION
END_FUNCTION_BLOCK

FUNCTION_BLOCK SmallSortingConveyor
VAR_INPUT
	Switch : Switch;
	Motor : Motor;	
	//Software
	SFCReset : BOOL;
	InitCompleted : BOOL;
	SC_Refill_AllowToOperate : BOOL; //SC=SeperatorConveyor
	AutomaticExecuteCompleted : BOOL;
	EmergencyHandeled : BOOL;
END_VAR
VAR_OUTPUT
	//Software
	SmallConveyor_IsSorting : BOOL;
	SmallConveyor_WPSorted : BOOL;
END_VAR
VAR		
	//Hardware
	SmallConveyor_Beginning_PresenceSensor AT %I* : BOOL;
	SmallConveyor_InductiveSensor AT %I* : BOOL;
	SmallConveyor_LightSensor AT %I* : BOOL;
	SmallConveyor_End_PresenceSensor AT %I* : BOOL;
	SmallConveyor_Ramp_PresenceSensor AT %I* : BOOL;
	
	//Software
	Timer : TON;
END_VAR

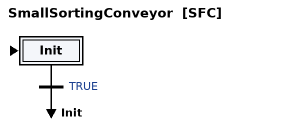
INITIAL_STEP Init:
END_STEP
TRANSITION FROM Init TO Init
  := TRUE;
END_TRANSITION

ACTION ACT_SortWP:
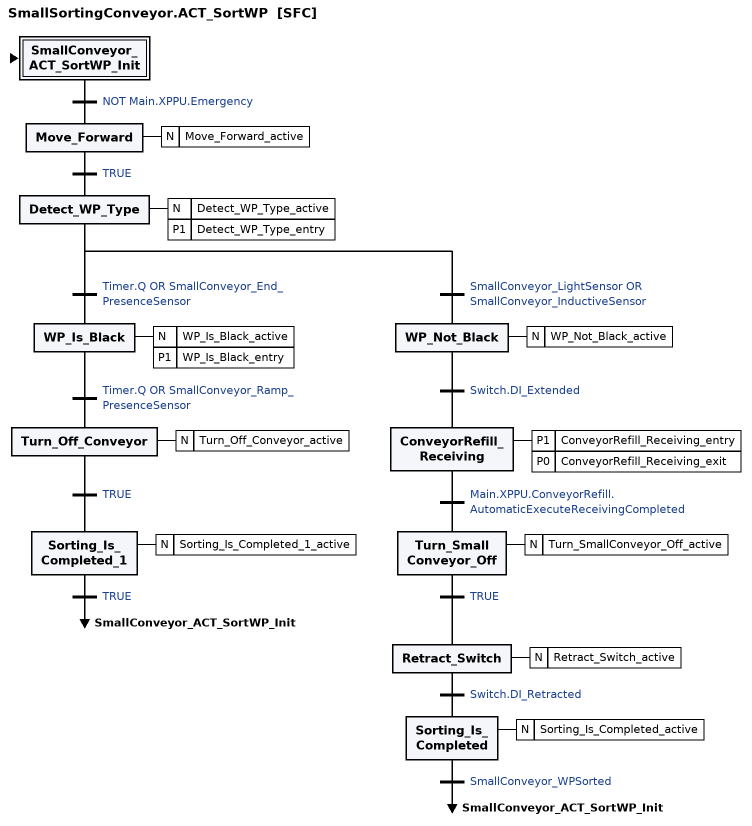
INITIAL_STEP SmallConveyor_ACT_SortWP_Init:
END_STEP
TRANSITION FROM SmallConveyor_ACT_SortWP_Init TO Move_Forward
  := NOT Main.XPPU.Emergency;
END_TRANSITION
STEP Move_Forward:
  Move_Forward_active(N);
END_STEP
TRANSITION FROM Move_Forward TO Detect_WP_Type
  := TRUE;
END_TRANSITION
STEP Detect_WP_Type:
  Detect_WP_Type_active(N);
  Detect_WP_Type_entry(P1);
END_STEP
TRANSITION FROM Detect_WP_Type TO WP_Is_Black
  := Timer.Q OR SmallConveyor_End_PresenceSensor;
END_TRANSITION
TRANSITION FROM Detect_WP_Type TO WP_Not_Black
  := SmallConveyor_LightSensor OR SmallConveyor_InductiveSensor;
END_TRANSITION
STEP WP_Is_Black:
  WP_Is_Black_active(N);
  WP_Is_Black_entry(P1);
END_STEP
TRANSITION FROM WP_Is_Black TO Turn_Off_Conveyor
  := Timer.Q OR SmallConveyor_Ramp_PresenceSensor;
END_TRANSITION
STEP Turn_Off_Conveyor:
  Turn_Off_Conveyor_active(N);
END_STEP
TRANSITION FROM Turn_Off_Conveyor TO Sorting_Is_Completed_1
  := TRUE;
END_TRANSITION
STEP Sorting_Is_Completed_1:
  Sorting_Is_Completed_1_active(N);
END_STEP
TRANSITION FROM Sorting_Is_Completed_1 TO SmallConveyor_ACT_SortWP_Init
  := TRUE;
END_TRANSITION
STEP WP_Not_Black:
  WP_Not_Black_active(N);
END_STEP
TRANSITION FROM WP_Not_Black TO ConveyorRefill_Receiving
  := Switch.DI_Extended;
END_TRANSITION
STEP ConveyorRefill_Receiving:
  ConveyorRefill_Receiving_entry(P1);
  ConveyorRefill_Receiving_exit(P0);
END_STEP
TRANSITION FROM ConveyorRefill_Receiving TO Turn_SmallConveyor_Off
  := Main.XPPU.ConveyorRefill.AutomaticExecuteReceivingCompleted;
END_TRANSITION
STEP Turn_SmallConveyor_Off:
  Turn_SmallConveyor_Off_active(N);
END_STEP
TRANSITION FROM Turn_SmallConveyor_Off TO Retract_Switch
  := TRUE;
END_TRANSITION
STEP Retract_Switch:
  Retract_Switch_active(N);
END_STEP
TRANSITION FROM Retract_Switch TO Sorting_Is_Completed
  := Switch.DI_Retracted;
END_TRANSITION
STEP Sorting_Is_Completed:
  Sorting_Is_Completed_active(N);
END_STEP
TRANSITION FROM Sorting_Is_Completed TO SmallConveyor_ACT_SortWP_Init
  := SmallConveyor_WPSorted;
END_TRANSITION
END_ACTION

ACTION ACT_AutomaticExecute:
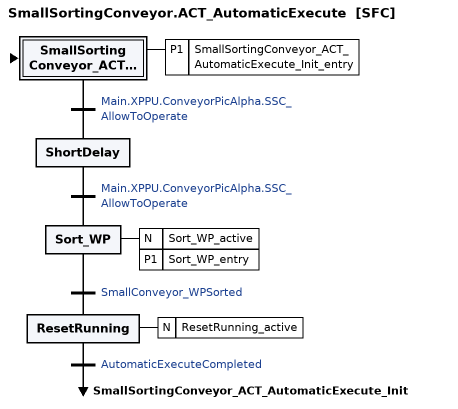
INITIAL_STEP SmallSortingConveyor_ACT_AutomaticExecute_Init:
  SmallSortingConveyor_ACT_AutomaticExecute_Init_entry(P1);
END_STEP
TRANSITION FROM SmallSortingConveyor_ACT_AutomaticExecute_Init TO ShortDelay
  := Main.XPPU.ConveyorPicAlpha.SSC_AllowToOperate;
END_TRANSITION
STEP ShortDelay:
END_STEP
TRANSITION FROM ShortDelay TO Sort_WP
  := Main.XPPU.ConveyorPicAlpha.SSC_AllowToOperate;
END_TRANSITION
STEP Sort_WP:
  Sort_WP_active(N);
  Sort_WP_entry(P1);
END_STEP
TRANSITION FROM Sort_WP TO ResetRunning
  := SmallConveyor_WPSorted;
END_TRANSITION
STEP ResetRunning:
  ResetRunning_active(N);
END_STEP
TRANSITION FROM ResetRunning TO SmallSortingConveyor_ACT_AutomaticExecute_Init
  := AutomaticExecuteCompleted;
END_TRANSITION
END_ACTION

ACTION ACT_Init:
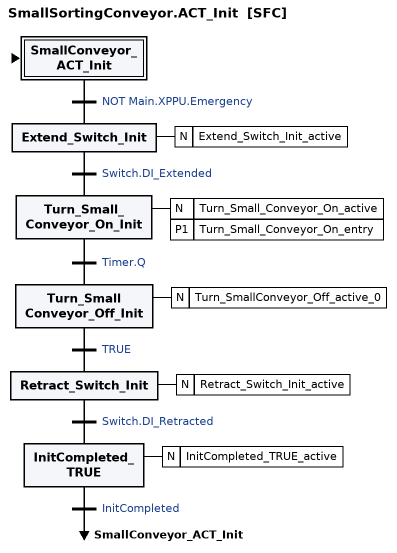
INITIAL_STEP SmallConveyor_ACT_Init:
END_STEP
TRANSITION FROM SmallConveyor_ACT_Init TO Extend_Switch_Init
  := NOT Main.XPPU.Emergency;
END_TRANSITION
STEP Extend_Switch_Init:
  Extend_Switch_Init_active(N);
END_STEP
TRANSITION FROM Extend_Switch_Init TO Turn_Small_Conveyor_On_Init
  := Switch.DI_Extended;
END_TRANSITION
STEP Turn_Small_Conveyor_On_Init:
  Turn_Small_Conveyor_On_active(N);
  Turn_Small_Conveyor_On_entry(P1);
END_STEP
TRANSITION FROM Turn_Small_Conveyor_On_Init TO Turn_SmallConveyor_Off_Init
  := Timer.Q;
END_TRANSITION
STEP Turn_SmallConveyor_Off_Init:
  Turn_SmallConveyor_Off_active_0(N);
END_STEP
TRANSITION FROM Turn_SmallConveyor_Off_Init TO Retract_Switch_Init
  := TRUE;
END_TRANSITION
STEP Retract_Switch_Init:
  Retract_Switch_Init_active(N);
END_STEP
TRANSITION FROM Retract_Switch_Init TO InitCompleted_TRUE
  := Switch.DI_Retracted;
END_TRANSITION
STEP InitCompleted_TRUE:
  InitCompleted_TRUE_active(N);
END_STEP
TRANSITION FROM InitCompleted_TRUE TO SmallConveyor_ACT_Init
  := InitCompleted;
END_TRANSITION
END_ACTION

ACTION ACT_EmergencyStop:
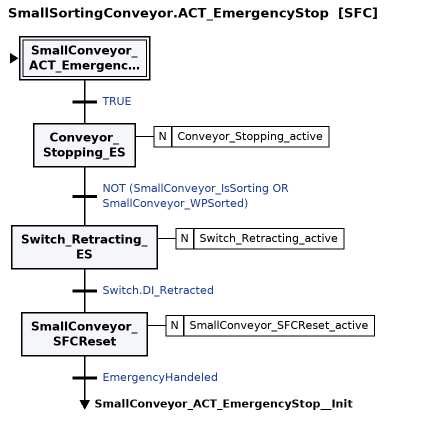
INITIAL_STEP SmallConveyor_ACT_EmergencyStop__Init:
END_STEP
TRANSITION FROM SmallConveyor_ACT_EmergencyStop__Init TO Conveyor_Stopping_ES
  := TRUE;
END_TRANSITION
STEP Conveyor_Stopping_ES:
  Conveyor_Stopping_active(N);
END_STEP
TRANSITION FROM Conveyor_Stopping_ES TO Switch_Retracting_ES
  := NOT (SmallConveyor_IsSorting OR SmallConveyor_WPSorted);
END_TRANSITION
STEP Switch_Retracting_ES:
  Switch_Retracting_active(N);
END_STEP
TRANSITION FROM Switch_Retracting_ES TO SmallConveyor_SFCReset
  := Switch.DI_Retracted;
END_TRANSITION
STEP SmallConveyor_SFCReset:
  SmallConveyor_SFCReset_active(N);
END_STEP
TRANSITION FROM SmallConveyor_SFCReset TO SmallConveyor_ACT_EmergencyStop__Init
  := EmergencyHandeled;
END_TRANSITION
END_ACTION

ACTION Move_Forward_active:
                      Motor.ACT_TurnForwards();
                    
END_ACTION

ACTION StartConveyor_active:
                      //Main.XPPU.ConveyorPicAlpha.ACT_MoveForwards();
Timer(IN:=TRUE, PT:=T#3S);
                    
END_ACTION

ACTION SmallConveyor_SFCReset_active:
                       EmergencyHandeled:=TRUE;	
                    
END_ACTION

ACTION Conveyor_Stopping_active:
                      SmallConveyor_IsSorting:=FALSE;
SmallConveyor_WPSorted:=FALSE;

Motor.ACT_Stop();
                    
END_ACTION

ACTION Detect_WP_Type_active:
                      Timer(IN:=TRUE, PT:=T#3000ms);
                    
END_ACTION

ACTION StartConveyor_entry:
                      Timer(IN:=FALSE);
                    
END_ACTION

ACTION Sort_WP_active:
                      ACT_SortWP();
                    
END_ACTION

ACTION HelpACT_WPSorted_FALSE:
                      SmallConveyor_WPSorted:=FALSE;
                    
END_ACTION

ACTION ResetRunning_active:
                      AutomaticExecuteCompleted:=TRUE;
                    
END_ACTION

ACTION Seperate_WP_active:
                      MAIN.XPPU.ConveyorRefill.ACT_SeperateWP();
                    
END_ACTION

ACTION ConveyorRefill_Receiving_entry:
                      SC_Refill_AllowToOperate:=TRUE;
                    
END_ACTION

ACTION StopConveyor_active:
                      //Main.XPPU.ConveyorPicAlpha.ACT_Stop();
                    
END_ACTION

ACTION ShortDelay_entry:
                      Timer(IN:=FALSE);
                    
END_ACTION

ACTION WP_Is_Black_active:
                      Timer(In:=TRUE, PT:=T#2000ms);
                    
END_ACTION

ACTION Turn_Refill_Conveyor_On_active:
                      //MAIN.XPPU.ConveyorRefill.ACT_MoveForwards();
                    
END_ACTION

ACTION Switch_Retracting_active:
                      Switch.ACT_Retract();
                    
END_ACTION

ACTION Stopping_WP_active:
                      Timer(IN:=TRUE, PT:=T#2000ms);
                    
END_ACTION

ACTION Extend_Switch_Init_active:
                      Switch.ACT_Extend();
                    
END_ACTION

ACTION Turn_RefillConveyor_Off_active:
                      //Main.XPPU.ConveyorRefill.ACT_Stop();
                    
END_ACTION

ACTION Count_Up_active:
                      
                    
END_ACTION

ACTION Retract_Switch_Init_active:
                      Switch.ACT_Retract();
                    
END_ACTION

ACTION Stopping_WP_entry:
                      Timer(IN:=FALSE);
                    
END_ACTION

ACTION Sorting_Is_Completed_exit:
                      SmallConveyor_IsSorting:=FALSE;
                    
END_ACTION

ACTION WP_Is_Black_entry:
                      Timer(In:=FALSE);
                    
END_ACTION

ACTION Turn_SmallConveyor_Off_active_0:
                      Motor.ACT_Stop();
                    
END_ACTION

ACTION Turn_Small_Conveyor_On_entry:
                      Timer(IN:=FALSE);
                    
END_ACTION

ACTION Sorting_Is_Completed_1_exit:
                      
                    
END_ACTION

ACTION Sorting_Is_Completed_1_active:
                      SmallConveyor_IsSorting:=FALSE;
SmallConveyor_WPSorted:=TRUE;
                    
END_ACTION

ACTION WP_From_ConveyorPicAlpha_active:
                      //MAIN.XPPU.ConveyorPicAlpha.ACT_MoveForwards();
Motor.ACT_TurnForwards();
                    
END_ACTION

ACTION Turn_Off_RefillConveyor_active:
                      //MAIN.XPPU.ConveyorRefill.ACT_Stop();
                    
END_ACTION

ACTION Turn_Refill_Conveyor_On_active_0:
                      //Main.XPPU.ConveyorRefill.ACT_MoveForwards();
                    
END_ACTION

ACTION ConveyorRefill_Receiving_exit:
                      SC_Refill_AllowToOperate:=FALSE;
                    
END_ACTION

ACTION Retract_Switch_active:
                      Switch.ACT_Retract();
                    
END_ACTION

ACTION Turn_SmallConveyor_Off_active:
                      Motor.ACT_Stop();
                    
END_ACTION

ACTION Turn_Small_Conveyor_On_active:
                      Motor.ACT_TurnForwards();
Timer(IN:=TRUE, PT:=T#2000ms);
                    
END_ACTION

ACTION ShortDelay_active:
                      Timer(IN:=TRUE, PT:=T#500ms);
                    
END_ACTION

ACTION WP_Not_Black_active:
                      Switch.ACT_Extend();
                    
END_ACTION

ACTION SmallSortingConveyor_ACT_AutomaticExecute_Init_entry:
                      AutomaticExecuteCompleted:=FALSE;
                    
END_ACTION

ACTION Detect_WP_Type_entry:
                      SmallConveyor_IsSorting:=TRUE;
SmallConveyor_WPSorted:=FALSE;
Timer(IN:=FALSE);
                    
END_ACTION

ACTION Count_WP_At_RefillConveyor_active:
                      
                    
END_ACTION

ACTION InitCompleted_FALSE_active:
                      InitCompleted:=FALSE;
                    
END_ACTION

ACTION Sort_WP_entry:
                      SmallConveyor_IsSorting:=TRUE;
SmallConveyor_WPSorted:=FALSE;
                    
END_ACTION

ACTION Turn_Off_Conveyor_active:
                      Motor.ACT_Stop();
                    
END_ACTION

ACTION Sorting_Is_Completed_active:
                      SmallConveyor_IsSorting:=FALSE;
SmallConveyor_WPSorted:=TRUE;
                    
END_ACTION

ACTION InitCompleted_TRUE_active:
                      InitCompleted:=TRUE;
                    
END_ACTION

ACTION Sort_WP_At_Conveyor_active:
                      MAIN.XPPU.LargeSortingConveyor.ACT_SortWP();
                    
END_ACTION
END_FUNCTION_BLOCK

FUNCTION_BLOCK Stack
VAR_INPUT	
	Seperator : MonostableCylinder;	
	//Software
	SFCReset : BOOL;
	InitCompleted : BOOL;
	EmergencyHandeled : BOOL;	
END_VAR
VAR_OUTPUT	
	//Software
	Stack_WPType_White : BOOL;
	Stack_WPType_Black : BOOL;
	Stack_WPType_Metallic : BOOL;
	Stack_WPWeight_Light : BOOL;
	Stack_WPWeight_Medium : BOOL;
	Stack_WPWeight_Heavy : BOOL;
	Stack_WPProvided : BOOL;	
END_VAR
VAR
	//Hardware
	Stack_WorkpieceReady AT %I* : BOOL;
	Stack_InductiveSensor AT %I* : BOOL;
	Stack_OpticalSensor AT %I* : BOOL;
	Stack_WPWeight AT %I* : INT;
	Stack_StartButton AT %I* : BOOL;
	Stack_EmergencyStop AT %I* : BOOL;	
	StackGreenLamp AT %Q* : BOOL;
	StackWhiteLamp AT %Q* : BOOL;
	
	//Software
	Timer : TON;		
END_VAR

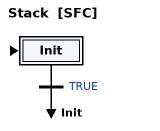
INITIAL_STEP Init:
END_STEP
TRANSITION FROM Init TO Init
  := TRUE;
END_TRANSITION

ACTION ACT_GreenLampOn:
                      StackGreenLamp:=TRUE;
                    
END_ACTION

ACTION ACT_GreenLampOff:
                      StackGreenLamp:=FALSE;
                    
END_ACTION

ACTION ACT_WhiteLampOff:
                      StackWhiteLamp:=FALSE;
                    
END_ACTION

ACTION ACT_WhiteLampOn:
                      StackWhiteLamp:=TRUE;
StackGreenLamp:=FALSE;
                    
END_ACTION

ACTION ACT_ProvideWP:
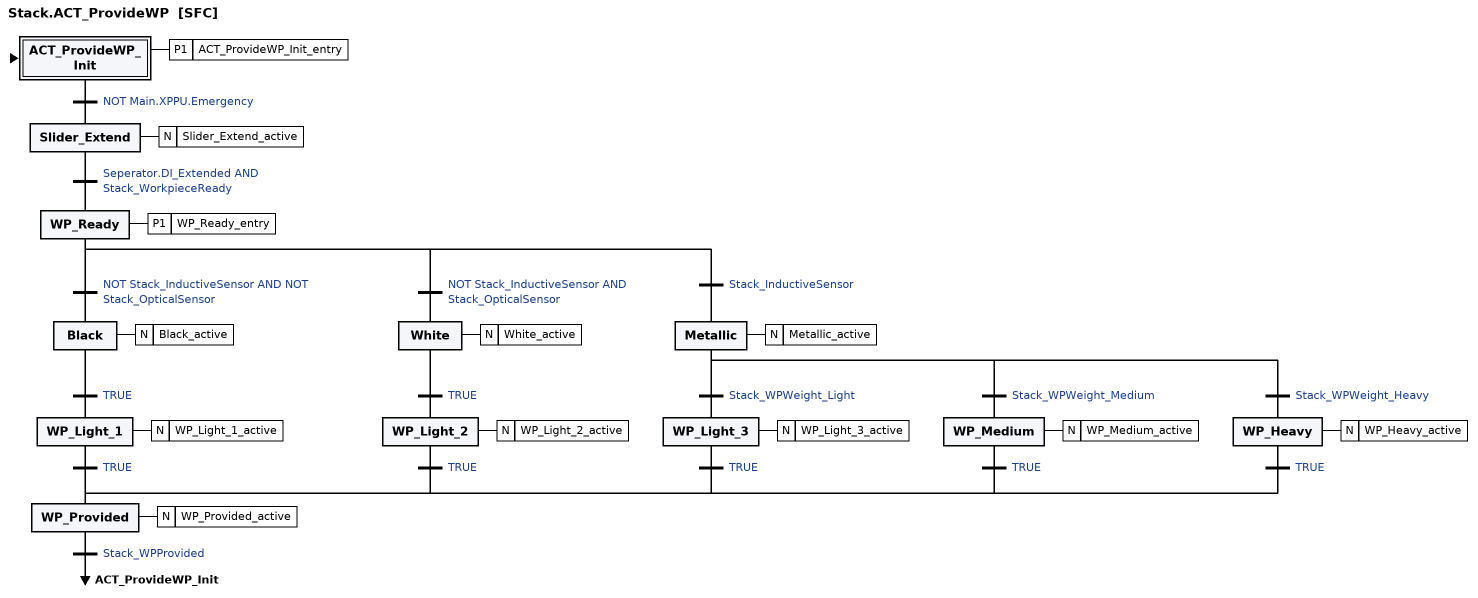
INITIAL_STEP ACT_ProvideWP_Init:
  ACT_ProvideWP_Init_entry(P1);
END_STEP
TRANSITION FROM ACT_ProvideWP_Init TO Slider_Extend
  := NOT Main.XPPU.Emergency;
END_TRANSITION
STEP Slider_Extend:
  Slider_Extend_active(N);
END_STEP
TRANSITION FROM Slider_Extend TO WP_Ready
  := Seperator.DI_Extended AND Stack_WorkpieceReady;
END_TRANSITION
STEP WP_Ready:
  WP_Ready_entry(P1);
END_STEP
TRANSITION FROM WP_Ready TO Black
  := NOT Stack_InductiveSensor AND NOT Stack_OpticalSensor;
END_TRANSITION
TRANSITION FROM WP_Ready TO White
  := NOT Stack_InductiveSensor AND Stack_OpticalSensor;
END_TRANSITION
TRANSITION FROM WP_Ready TO Metallic
  := Stack_InductiveSensor;
END_TRANSITION
STEP Black:
  Black_active(N);
END_STEP
TRANSITION FROM Black TO WP_Light_1
  := TRUE;
END_TRANSITION
STEP WP_Light_1:
  WP_Light_1_active(N);
END_STEP
TRANSITION FROM WP_Light_1 TO WP_Provided
  := TRUE;
END_TRANSITION
STEP White:
  White_active(N);
END_STEP
TRANSITION FROM White TO WP_Light_2
  := TRUE;
END_TRANSITION
STEP WP_Light_2:
  WP_Light_2_active(N);
END_STEP
TRANSITION FROM WP_Light_2 TO WP_Provided
  := TRUE;
END_TRANSITION
STEP Metallic:
  Metallic_active(N);
END_STEP
TRANSITION FROM Metallic TO WP_Light_3
  := Stack_WPWeight_Light;
END_TRANSITION
TRANSITION FROM Metallic TO WP_Medium
  := Stack_WPWeight_Medium;
END_TRANSITION
TRANSITION FROM Metallic TO WP_Heavy
  := Stack_WPWeight_Heavy;
END_TRANSITION
STEP WP_Light_3:
  WP_Light_3_active(N);
END_STEP
TRANSITION FROM WP_Light_3 TO WP_Provided
  := TRUE;
END_TRANSITION
STEP WP_Medium:
  WP_Medium_active(N);
END_STEP
TRANSITION FROM WP_Medium TO WP_Provided
  := TRUE;
END_TRANSITION
STEP WP_Heavy:
  WP_Heavy_active(N);
END_STEP
TRANSITION FROM WP_Heavy TO WP_Provided
  := TRUE;
END_TRANSITION
STEP WP_Provided:
  WP_Provided_active(N);
END_STEP
TRANSITION FROM WP_Provided TO ACT_ProvideWP_Init
  := Stack_WPProvided;
END_TRANSITION
END_ACTION

ACTION Slider_Extend_active:
                      Seperator.ACT_Extend();
                    
END_ACTION

ACTION Crane_To_Magazine_active:
                      Main.XPPU.Crane.ACT_MoveToStack();
                    
END_ACTION

ACTION Provide_WP_active:
                      ACT_ProvideWP();
                    
END_ACTION

ACTION WP_Ready_entry:
                      Stack_WPType_White:=FALSE;
Stack_WPType_Black:=FALSE;
Stack_WPType_Metallic:=FALSE;
Stack_WPWeight_Light:=FALSE;
Stack_WPWeight_Medium:=FALSE;
Stack_WPWeight_Heavy:=FALSE;
                    
END_ACTION

ACTION Stack_Retracing_active:
                      Seperator.ACT_Retract();
                    
END_ACTION

ACTION Short_Delay_active:
                      Timer(IN:=TRUE, PT:=T#50ms);
                    
END_ACTION

ACTION Slider_Move_In_active:
                      Seperator.ACT_Retract();
                    
END_ACTION

ACTION Short_Delay_entry:
                      Timer(IN:=FALSE);
                    
END_ACTION

ACTION WP_Heavy_active:
                      Stack_WPWeight_Heavy:=TRUE;
                    
END_ACTION

ACTION WP_Light_2_active:
                      Stack_WPWeight_Light:=TRUE;
                    
END_ACTION

ACTION Set_WP_Parameters_active:
                      IF(NOT Stack_InductiveSensor AND NOT Stack_OpticalSensor)THEN
	Stack_WPType_Black:=TRUE;
	Stack_WPType_White:=FALSE;
	Stack_WPType_Metallic:=FALSE;
ELSIF(NOT Stack_InductiveSensor AND Stack_OpticalSensor)THEN
	Stack_WPType_Black:=FALSE;
	Stack_WPType_White:=TRUE;
	Stack_WPType_Metallic:=FALSE;
ELSIF(Stack_InductiveSensor)THEN
	Stack_WPType_Black:=FALSE;
	Stack_WPType_White:=FALSE;
	Stack_WPType_Metallic:=TRUE;
END_IF

IF(Stack_WPType_Black OR Stack_WPType_White OR(Stack_WPType_Metallic AND Stack_WPWeight < 12000))THEN
	Stack_WPWeight_Light:=TRUE;
	Stack_WPWeight_Medium:=FALSE;
	Stack_WPWeight_Heavy:=FALSE;
ELSIF(12000<Stack_WPWeight AND Stack_WPWeight<=24000)THEN
	Stack_WPWeight_Light:=FALSE;
	Stack_WPWeight_Medium:=TRUE;
	Stack_WPWeight_Heavy:=FALSE;	
ELSIF(24000<=Stack_WPWeight)THEN
	Stack_WPWeight_Light:=FALSE;
	Stack_WPWeight_Medium:=FALSE;
	Stack_WPWeight_Heavy:=TRUE;	
END_IF

Stack_WPProvided:=TRUE;
                    
END_ACTION

ACTION Metallic_active:
                      Stack_WPType_Metallic:=TRUE;
IF(Stack_WPWeight < 12000)THEN
	Stack_WPWeight_Light:=TRUE;
END_IF
IF(12000<Stack_WPWeight AND Stack_WPWeight<=24000)THEN
	Stack_WPWeight_Medium:=TRUE;
END_IF
IF(24000<=Stack_WPWeight)THEN
	Stack_WPWeight_Heavy:=TRUE;
END_IF

                    
END_ACTION

ACTION WP_Allreday_Provided_active:
                      
                    
END_ACTION

ACTION PutDown_WP_active:
                      Main.XPPU.Crane.ACT_PutDownWP();
                    
END_ACTION

ACTION Stack_SFCReset_active:
                       EmergencyHandeled:=TRUE;		
                    
END_ACTION

ACTION Magazine_ACT_EmergencyStop_Init_entry:
                      StackGreenLamp:=FALSE;
StackWhiteLamp:=FALSE;
                    
END_ACTION

ACTION WP_Provided_active:
                      Stack_WPProvided:=TRUE;
                    
END_ACTION

ACTION WP_Light_1_active:
                      Stack_WPWeight_Light:=TRUE;
                    
END_ACTION

ACTION Black_active:
                      Stack_WPType_Black:=TRUE;
                    
END_ACTION

ACTION InitCompleted_TRUE_active:
                      InitCompleted:=TRUE;
                    
END_ACTION

ACTION Stack_ACT_Init_entry:
                      

                    
END_ACTION

ACTION WP_Light_3_active:
                      Stack_WPWeight_Light:=TRUE;
                    
END_ACTION

ACTION WP_Medium_active:
                      Stack_WPWeight_Medium:=TRUE;
                    
END_ACTION

ACTION Slider_Move_In_2_active:
                      Seperator.ACT_Retract();
                    
END_ACTION

ACTION WP_To_Conveyor_active:
                      Main.XPPU.Crane.ACT_MoveToConveyor();
                    
END_ACTION

ACTION Stack_Retracting_active:
                      Stack_WPType_White:=FALSE;
Stack_WPType_Black:=FALSE;
Stack_WPType_Metallic:=FALSE;
Stack_WPWeight_Light:=FALSE;
Stack_WPWeight_Medium:=FALSE;
Stack_WPWeight_Heavy:=FALSE;
Stack_WPProvided:=FALSE;

Seperator.ACT_Retract();
                    
END_ACTION

ACTION SortWP_Init_active:
                      Main.XPPU.LargeSortingConveyor.ACT_SortWP();
                    
END_ACTION

ACTION Pick_Up_WP_active:
                      Main.XPPU.Crane.ACT_PickUpWP();
                    
END_ACTION

ACTION White_active:
                      Stack_WPType_White:=TRUE;
                    
END_ACTION

ACTION Retract_Cylinder_Init_active:
                      Seperator.ACT_Retract();
                    
END_ACTION

ACTION ACT_ProvideWP_Init_entry:
                      Stack_WPProvided:=FALSE;
                    
END_ACTION

ACTION ACT_EmergencyStop:
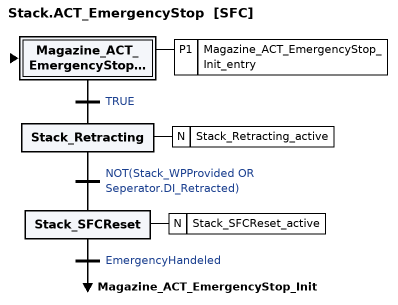
INITIAL_STEP Magazine_ACT_EmergencyStop_Init:
  Magazine_ACT_EmergencyStop_Init_entry(P1);
END_STEP
TRANSITION FROM Magazine_ACT_EmergencyStop_Init TO Stack_Retracting
  := TRUE;
END_TRANSITION
STEP Stack_Retracting:
  Stack_Retracting_active(N);
END_STEP
TRANSITION FROM Stack_Retracting TO Stack_SFCReset
  := NOT(Stack_WPProvided OR Seperator.DI_Retracted);
END_TRANSITION
STEP Stack_SFCReset:
  Stack_SFCReset_active(N);
END_STEP
TRANSITION FROM Stack_SFCReset TO Magazine_ACT_EmergencyStop_Init
  := EmergencyHandeled;
END_TRANSITION
END_ACTION

ACTION ACT_AutomaticExecute:
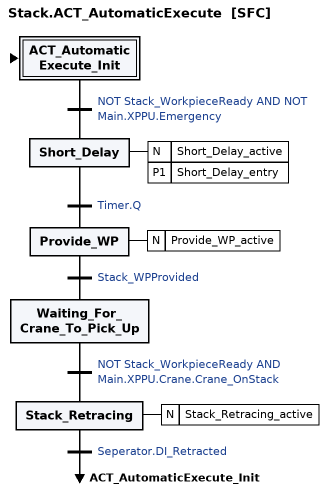
INITIAL_STEP ACT_AutomaticExecute_Init:
END_STEP
TRANSITION FROM ACT_AutomaticExecute_Init TO Short_Delay
  := NOT Stack_WorkpieceReady AND NOT Main.XPPU.Emergency;
END_TRANSITION
STEP Short_Delay:
  Short_Delay_active(N);
  Short_Delay_entry(P1);
END_STEP
TRANSITION FROM Short_Delay TO Provide_WP
  := Timer.Q;
END_TRANSITION
STEP Provide_WP:
  Provide_WP_active(N);
END_STEP
TRANSITION FROM Provide_WP TO Waiting_For_Crane_To_Pick_Up
  := Stack_WPProvided;
END_TRANSITION
STEP Waiting_For_Crane_To_Pick_Up:
END_STEP
TRANSITION FROM Waiting_For_Crane_To_Pick_Up TO Stack_Retracing
  := NOT Stack_WorkpieceReady AND Main.XPPU.Crane.Crane_OnStack;
END_TRANSITION
STEP Stack_Retracing:
  Stack_Retracing_active(N);
END_STEP
TRANSITION FROM Stack_Retracing TO ACT_AutomaticExecute_Init
  := Seperator.DI_Retracted;
END_TRANSITION
END_ACTION

ACTION ACT_Init:
